  MoveL 2621 to (-2.16, 59.3, -119.45) mm, rotated rx 105.8 ry 33.04 rz -145.95 deg; joints [-4.768, -29.357, 102.728, 146.483, 85.031, 18.435, -295]
  MoveL 2622 to (0.51, 59.77, -119.55) mm, rotated rx 105.8 ry 33.04 rz -145.95 deg; joints [-4.771, -29.24, 102.473, 146.472, 84.917, 18.512, -295]
  MoveL 2623 to (2.52, 60.11, -119.76) mm, rotated rx 105.8 ry 33.04 rz -145.95 deg; joints [-4.779, -29.151, 102.281, 146.459, 84.832, 18.572, -295]
  MoveL 2624 to (4.69, 60.48, -119.96) mm, rotated rx 105.8 ry 33.04 rz -145.95 deg; joints [-4.787, -29.055, 102.073, 146.446, 84.74, 18.636, -295]
  MoveL 2625 to (6.69, 60.8, -120.25) mm, rotated rx 105.8 ry 33.04 rz -145.95 deg; joints [-4.798, -28.966, 101.881, 146.43, 84.657, 18.695, -295]
  MoveL 2626 to (8.64, 61.14, -120.38) mm, rotated rx 105.8 ry 33.04 rz -145.95 deg; joints [-4.803, -28.879, 101.693, 146.42, 84.573, 18.753, -295]
  MoveL 2627 to (10.7, 61.51, -120.39) mm, rotated rx 105.8 ry 33.04 rz -145.95 deg; joints [-4.803, -28.789, 101.495, 146.414, 84.483, 18.813, -295]
  MoveL 2628 to (12.45, 61.78, -120.62) mm, rotated rx 105.8 ry 33.04 rz -145.95 deg; joints [-4.812, -28.709, 101.326, 146.401, 84.41, 18.864, -295]
  Set speed (1000.0 mm/s)
  MoveL 2629 to (33.8, 76.72, -120.62) mm, rotated rx 105.8 ry 33.04 rz -145.95 deg; joints [-4.805, -28.216, 99.114, 146.302, 82.978, 19.821, -295]
  Set speed (1000.0 mm/s)
  MoveL 2630 to (37.55, 71.37, -131.81) mm, rotated rx 105.8 ry 33.04 rz -145.95 deg; joints [-5.233, -27.799, 98.812, 145.891, 83.151, 19.873, -295]
  Set speed (100.0 mm/s)
  MoveL 2631 to (21.02, 59.8, -131.81) mm, rotated rx 105.8 ry 33.04 rz -145.95 deg; joints [-5.244, -28.182, 100.529, 145.963, 84.258, 19.124, -295]
  MoveL 2632 to (18.89, 59.68, -131.81) mm, rotated rx 105.8 ry 33.04 rz -145.95 deg; joints [-5.245, -28.288, 100.733, 145.968, 84.339, 19.069, -295]
  MoveL 2633 to (16.66, 59.58, -131.71) mm, rotated rx 105.8 ry 33.04 rz -145.95 deg; joints [-5.242, -28.4, 100.946, 145.976, 84.423, 19.012, -295]
  MoveL 2634 to (14.32, 59.52, -131.42) mm, rotated rx 105.8 ry 33.04 rz -145.95 deg; joints [-5.231, -28.519, 101.169, 145.992, 84.508, 18.95, -295]
  MoveL 2635 to (12.07, 59.46, -131.07) mm, rotated rx 105.8 ry 33.04 rz -145.95 deg; joints [-5.218, -28.633, 101.383, 146.01, 84.588, 18.891, -295]
  MoveL 2636 to (10, 59.38, -130.88) mm, rotated rx 105.8 ry 33.04 rz -145.95 deg; joints [-5.212, -28.737, 101.579, 146.022, 84.664, 18.837, -295]
  MoveL 2637 to (8.05, 59.28, -130.75) mm, rotated rx 105.8 ry 33.04 rz -145.95 deg; joints [-5.207, -28.833, 101.764, 146.031, 84.736, 18.787, -295]
  MoveL 2638 to (6, 59.18, -130.7) mm, rotated rx 105.8 ry 33.04 rz -145.95 deg; joints [-5.206, -28.935, 101.959, 146.037, 84.813, 18.734, -295]
  MoveL 2639 to (3.87, 59.06, -130.68) mm, rotated rx 105.8 ry 33.04 rz -145.95 deg; joints [-5.205, -29.04, 102.16, 146.042, 84.893, 18.68, -295]
  MoveL 2640 to (1.75, 58.95, -130.56) mm, rotated rx 105.8 ry 33.04 rz -145.95 deg; joints [-5.201, -29.144, 102.361, 146.051, 84.972, 18.625, -295]
  MoveL 2641 to (-0.53, 58.83, -130.3) mm, rotated rx 105.8 ry 33.04 rz -145.95 deg; joints [-5.192, -29.257, 102.576, 146.065, 85.056, 18.565, -295]
  MoveL 2642 to (-2.93, 58.7, -130.11) mm, rotated rx 105.8 ry 33.04 rz -145.95 deg; joints [-5.185, -29.374, 102.802, 146.077, 85.145, 18.503, -295]
  MoveL 2643 to (-5.26, 58.57, -129.91) mm, rotated rx 105.8 ry 33.04 rz -145.95 deg; joints [-5.178, -29.488, 103.021, 146.089, 85.231, 18.442, -295]
  MoveL 2644 to (-7.39, 58.44, -129.8) mm, rotated rx 105.8 ry 33.04 rz -145.95 deg; joints [-5.174, -29.592, 103.221, 146.097, 85.31, 18.388, -295]
  MoveL 2645 to (-11.61, 58.19, -129.52) mm, rotated rx 105.8 ry 33.04 rz -145.95 deg; joints [-5.165, -29.797, 103.616, 146.115, 85.467, 18.279, -295]
  MoveL 2646 to (-13.78, 58.06, -129.46) mm, rotated rx 105.8 ry 33.04 rz -145.95 deg; joints [-5.163, -29.902, 103.819, 146.121, 85.547, 18.224, -295]
  MoveL 2647 to (-15.91, 57.92, -129.24) mm, rotated rx 105.8 ry 33.04 rz -145.95 deg; joints [-5.154, -30.004, 104.017, 146.133, 85.626, 18.168, -295]
  MoveL 2648 to (-18.01, 57.77, -129.08) mm, rotated rx 105.8 ry 33.04 rz -145.95 deg; joints [-5.149, -30.105, 104.214, 146.143, 85.704, 18.114, -295]
  MoveL 2649 to (-20.12, 57.62, -128.89) mm, rotated rx 105.8 ry 33.04 rz -145.95 deg; joints [-5.142, -30.206, 104.41, 146.153, 85.783, 18.059, -295]
  MoveL 2650 to (-22.29, 57.49, -128.8) mm, rotated rx 105.8 ry 33.04 rz -145.95 deg; joints [-5.139, -30.31, 104.611, 146.16, 85.863, 18.004, -295]
  MoveL 2651 to (-24.56, 57.32, -128.67) mm, rotated rx 105.8 ry 33.04 rz -145.95 deg; joints [-5.134, -30.418, 104.822, 146.169, 85.948, 17.945, -295]
  MoveL 2652 to (-26.46, 57.22, -128.61) mm, rotated rx 105.8 ry 33.04 rz -145.95 deg; joints [-5.132, -30.51, 104.998, 146.174, 86.017, 17.898, -295]
  MoveL 2653 to (-26.42, 56.56, -127.73) mm, rotated rx 105.8 ry 33.04 rz -145.95 deg; joints [-5.098, -30.478, 105.002, 146.209, 86.042, 17.87, -295]
  MoveL 2654 to (-26.12, 56.36, -127.32) mm, rotated rx 105.8 ry 33.04 rz -145.95 deg; joints [-5.081, -30.454, 104.977, 146.226, 86.038, 17.867, -295]
  MoveL 2655 to (-26.09, 56.3, -127.04) mm, rotated rx 105.8 ry 33.04 rz -145.95 deg; joints [-5.07, -30.449, 104.975, 146.236, 86.039, 17.863, -295]
  MoveL 2656 to (-26.4, 56.42, -126.92) mm, rotated rx 105.8 ry 33.04 rz -145.95 deg; joints [-5.066, -30.47, 105.002, 146.241, 86.043, 17.859, -295]
  MoveL 2657 to (-26.8, 56.62, -126.86) mm, rotated rx 105.8 ry 33.04 rz -145.95 deg; joints [-5.063, -30.5, 105.037, 146.244, 86.048, 17.855, -295]
  MoveL 2658 to (-27.3, 56.88, -126.83) mm, rotated rx 105.8 ry 33.04 rz -145.95 deg; joints [-5.062, -30.537, 105.08, 146.245, 86.052, 17.852, -295]
  MoveL 2659 to (-27.91, 57.21, -126.79) mm, rotated rx 105.8 ry 33.04 rz -145.95 deg; joints [-5.06, -30.582, 105.132, 146.247, 86.057, 17.848, -295]
  MoveL 2660 to (-28.46, 57.53, -126.76) mm, rotated rx 105.8 ry 33.04 rz -145.95 deg; joints [-5.059, -30.624, 105.179, 146.248, 86.062, 17.845, -295]
  MoveL 2661 to (-28.91, 57.79, -126.76) mm, rotated rx 105.8 ry 33.04 rz -145.95 deg; joints [-5.059, -30.659, 105.218, 146.249, 86.065, 17.843, -295]
  MoveL 2662 to (-29.34, 58.03, -126.75) mm, rotated rx 105.8 ry 33.04 rz -145.95 deg; joints [-5.058, -30.691, 105.254, 146.249, 86.068, 17.84, -295]
  MoveL 2663 to (-30.26, 58.51, -126.67) mm, rotated rx 105.8 ry 33.04 rz -145.95 deg; joints [-5.055, -30.76, 105.333, 146.253, 86.076, 17.833, -295]
  MoveL 2664 to (-30.76, 58.77, -126.62) mm, rotated rx 105.8 ry 33.04 rz -145.95 deg; joints [-5.053, -30.797, 105.376, 146.255, 86.081, 17.83, -295]
  MoveL 2665 to (-31.22, 58.99, -126.55) mm, rotated rx 105.8 ry 33.04 rz -145.95 deg; joints [-5.05, -30.83, 105.416, 146.258, 86.086, 17.825, -295]
  MoveL 2666 to (-31.64, 59.18, -126.48) mm, rotated rx 105.8 ry 33.04 rz -145.95 deg; joints [-5.047, -30.86, 105.452, 146.261, 86.091, 17.821, -295]
  MoveL 2667 to (-32.06, 59.39, -126.42) mm, rotated rx 105.8 ry 33.04 rz -145.95 deg; joints [-5.045, -30.89, 105.488, 146.264, 86.096, 17.817, -295]
  MoveL 2668 to (-32.48, 59.61, -126.39) mm, rotated rx 105.8 ry 33.04 rz -145.95 deg; joints [-5.044, -30.922, 105.525, 146.265, 86.099, 17.814, -295]
  MoveL 2669 to (-32.94, 59.87, -126.37) mm, rotated rx 105.8 ry 33.04 rz -145.95 deg; joints [-5.043, -30.956, 105.564, 146.266, 86.103, 17.812, -295]
  MoveL 2670 to (-36.09, 61.74, -126.37) mm, rotated rx 105.8 ry 33.04 rz -145.95 deg; joints [-5.042, -31.2, 105.831, 146.268, 86.122, 17.799, -295]
  MoveL 2671 to (-37.43, 62.66, -126.39) mm, rotated rx 105.8 ry 33.04 rz -145.95 deg; joints [-5.043, -31.31, 105.942, 146.267, 86.124, 17.798, -295]
  MoveL 2672 to (-37.85, 63.06, -126.42) mm, rotated rx 105.8 ry 33.04 rz -145.95 deg; joints [-5.044, -31.349, 105.976, 146.266, 86.12, 17.801, -295]
  MoveL 2673 to (-38.11, 63.42, -126.45) mm, rotated rx 105.8 ry 33.04 rz -145.95 deg; joints [-5.045, -31.378, 105.995, 146.264, 86.112, 17.807, -295]
  MoveL 2674 to (-38.23, 63.73, -126.49) mm, rotated rx 105.8 ry 33.04 rz -145.95 deg; joints [-5.047, -31.398, 106.003, 146.262, 86.101, 17.814, -295]
  MoveL 2675 to (-38.24, 63.88, -126.52) mm, rotated rx 105.8 ry 33.04 rz -145.95 deg; joints [-5.048, -31.406, 106.002, 146.261, 86.095, 17.819, -295]
  MoveL 2676 to (-38.22, 64.02, -126.54) mm, rotated rx 105.8 ry 33.04 rz -145.95 deg; joints [-5.048, -31.411, 105.999, 146.26, 86.088, 17.824, -295]
  MoveL 2677 to (-38.17, 64.15, -126.57) mm, rotated rx 105.8 ry 33.04 rz -145.95 deg; joints [-5.049, -31.414, 105.993, 146.259, 86.08, 17.829, -295]
  MoveL 2678 to (-38.1, 64.27, -126.6) mm, rotated rx 105.8 ry 33.04 rz -145.95 deg; joints [-5.051, -31.416, 105.985, 146.257, 86.072, 17.835, -295]
  MoveL 2679 to (-37.87, 64.49, -126.66) mm, rotated rx 105.8 ry 33.04 rz -145.95 deg; joints [-5.053, -31.414, 105.962, 146.254, 86.055, 17.847, -295]
  MoveL 2680 to (-37.16, 64.85, -126.79) mm, rotated rx 105.8 ry 33.04 rz -145.95 deg; joints [-5.058, -31.394, 105.893, 146.248, 86.015, 17.876, -295]
  MoveL 2681 to (-36.19, 65.11, -126.93) mm, rotated rx 105.8 ry 33.04 rz -145.95 deg; joints [-5.063, -31.357, 105.801, 146.24, 85.971, 17.907, -295]
  MoveL 2682 to (-33.87, 65.41, -127.2) mm, rotated rx 105.8 ry 33.04 rz -145.95 deg; joints [-5.073, -31.252, 105.586, 146.226, 85.88, 17.971, -295]
  MoveL 2683 to (-31.46, 65.57, -127.44) mm, rotated rx 105.8 ry 33.04 rz -145.95 deg; joints [-5.082, -31.137, 105.364, 146.213, 85.793, 18.032, -295]
  MoveL 2684 to (22.43, 68.71, -132.52) mm, rotated rx 105.8 ry 33.04 rz -145.95 deg; joints [-5.266, -28.487, 100.293, 145.91, 83.814, 19.434, -295]
  MoveL 2685 to (26.26, 68.94, -132.88) mm, rotated rx 105.8 ry 33.04 rz -145.95 deg; joints [-5.279, -28.295, 99.925, 145.887, 83.67, 19.537, -295]
  MoveL 2686 to (30.01, 68.97, -133.3) mm, rotated rx 105.8 ry 33.04 rz -145.95 deg; joints [-5.294, -28.099, 99.565, 145.862, 83.537, 19.633, -295]
  MoveL 2687 to (31.47, 68.71, -133.51) mm, rotated rx 105.8 ry 33.04 rz -145.95 deg; joints [-5.301, -28.01, 99.426, 145.851, 83.497, 19.664, -295]
  MoveL 2688 to (31.97, 68.47, -133.6) mm, rotated rx 105.8 ry 33.04 rz -145.95 deg; joints [-5.305, -27.974, 99.382, 145.847, 83.491, 19.67, -295]
  MoveL 2689 to (32.13, 68.32, -133.65) mm, rotated rx 105.8 ry 33.04 rz -145.95 deg; joints [-5.307, -27.959, 99.368, 145.845, 83.492, 19.67, -295]
  MoveL 2690 to (32.24, 68.14, -133.69) mm, rotated rx 105.8 ry 33.04 rz -145.95 deg; joints [-5.308, -27.946, 99.359, 145.844, 83.496, 19.667, -295]
  MoveL 2691 to (32.29, 67.94, -133.73) mm, rotated rx 105.8 ry 33.04 rz -145.95 deg; joints [-5.31, -27.935, 99.357, 145.843, 83.504, 19.663, -295]
  MoveL 2692 to (32.26, 67.71, -133.76) mm, rotated rx 105.8 ry 33.04 rz -145.95 deg; joints [-5.311, -27.927, 99.362, 145.843, 83.515, 19.655, -295]
  MoveL 2693 to (32.16, 67.45, -133.79) mm, rotated rx 105.8 ry 33.04 rz -145.95 deg; joints [-5.313, -27.921, 99.375, 145.842, 83.53, 19.646, -295]
  MoveL 2694 to (31.99, 67.16, -133.82) mm, rotated rx 105.8 ry 33.04 rz -145.95 deg; joints [-5.314, -27.918, 99.395, 145.843, 83.55, 19.633, -295]
  MoveL 2695 to (30.39, 65.66, -133.87) mm, rotated rx 105.8 ry 33.04 rz -145.95 deg; joints [-5.317, -27.939, 99.566, 145.849, 83.674, 19.549, -295]
  MoveL 2696 to (28.72, 64.39, -133.87) mm, rotated rx 105.8 ry 33.04 rz -145.95 deg; joints [-5.318, -27.974, 99.74, 145.856, 83.79, 19.471, -295]
  MoveL 2697 to (25.42, 62.49, -133.91) mm, rotated rx 105.8 ry 33.04 rz -145.95 deg; joints [-5.322, -28.067, 100.077, 145.867, 83.993, 19.334, -295]
  MoveL 2698 to (22.04, 61.43, -134.02) mm, rotated rx 105.8 ry 33.04 rz -145.95 deg; joints [-5.328, -28.199, 100.412, 145.873, 84.162, 19.221, -295]
  MoveL 2699 to (16, 61.08, -134.32) mm, rotated rx 105.8 ry 33.04 rz -145.95 deg; joints [-5.342, -28.499, 100.99, 145.875, 84.394, 19.068, -295]
  MoveL 2700 to (13.67, 61.43, -134.45) mm, rotated rx 105.8 ry 33.04 rz -145.95 deg; joints [-5.347, -28.636, 101.207, 145.874, 84.462, 19.024, -295]
  MoveL 2701 to (-20.45, 68.13, -136.31) mm, rotated rx 105.8 ry 33.04 rz -145.95 deg; joints [-5.429, -30.689, 104.317, 145.847, 85.349, 18.449, -295]
  MoveL 2702 to (-23.37, 68.69, -136.48) mm, rotated rx 105.8 ry 33.04 rz -145.95 deg; joints [-5.436, -30.864, 104.578, 145.844, 85.422, 18.401, -295]
  MoveL 2703 to (-27.1, 68.94, -136.72) mm, rotated rx 105.8 ry 33.04 rz -145.95 deg; joints [-5.447, -31.066, 104.918, 145.839, 85.537, 18.326, -295]
  MoveL 2704 to (-28.56, 68.71, -136.86) mm, rotated rx 105.8 ry 33.04 rz -145.95 deg; joints [-5.454, -31.131, 105.054, 145.836, 85.598, 18.287, -295]
  MoveL 2705 to (-29.05, 68.47, -136.93) mm, rotated rx 105.8 ry 33.04 rz -145.95 deg; joints [-5.457, -31.145, 105.102, 145.835, 85.626, 18.269, -295]
  MoveL 2706 to (-29.22, 68.32, -136.96) mm, rotated rx 105.8 ry 33.04 rz -145.95 deg; joints [-5.459, -31.147, 105.119, 145.834, 85.639, 18.261, -295]
  MoveL 2707 to (-29.33, 68.14, -137) mm, rotated rx 105.8 ry 33.04 rz -145.95 deg; joints [-5.46, -31.144, 105.131, 145.833, 85.651, 18.253, -295]
  MoveL 2708 to (-29.37, 67.93, -137.03) mm, rotated rx 105.8 ry 33.04 rz -145.95 deg; joints [-5.462, -31.137, 105.137, 145.832, 85.662, 18.246, -295]
  MoveL 2709 to (-29.34, 67.7, -137.07) mm, rotated rx 105.8 ry 33.04 rz -145.95 deg; joints [-5.463, -31.126, 105.137, 145.831, 85.672, 18.24, -295]
  MoveL 2710 to (-29.24, 67.44, -137.1) mm, rotated rx 105.8 ry 33.04 rz -145.95 deg; joints [-5.465, -31.109, 105.131, 145.83, 85.681, 18.234, -295]
  MoveL 2711 to (-29.06, 67.14, -137.14) mm, rotated rx 105.8 ry 33.04 rz -145.95 deg; joints [-5.466, -31.087, 105.118, 145.829, 85.689, 18.23, -295]
  MoveL 2712 to (-27.45, 65.66, -137.26) mm, rotated rx 105.8 ry 33.04 rz -145.95 deg; joints [-5.471, -30.939, 104.987, 145.825, 85.704, 18.221, -295]
  MoveL 2713 to (-27.03, 65.35, -137.28) mm, rotated rx 105.8 ry 33.04 rz -145.95 deg; joints [-5.472, -30.904, 104.952, 145.824, 85.704, 18.221, -295]
  MoveL 2714 to (-26.65, 65.1, -137.33) mm, rotated rx 105.8 ry 33.04 rz -145.95 deg; joints [-5.474, -30.873, 104.92, 145.822, 85.703, 18.222, -295]
  MoveL 2715 to (-26.27, 64.88, -137.4) mm, rotated rx 105.8 ry 33.04 rz -145.95 deg; joints [-5.477, -30.843, 104.888, 145.819, 85.701, 18.225, -295]
  MoveL 2716 to (-25.9, 64.64, -137.46) mm, rotated rx 105.8 ry 33.04 rz -145.95 deg; joints [-5.479, -30.814, 104.856, 145.817, 85.7, 18.226, -295]
  MoveL 2717 to (-25.51, 64.37, -137.49) mm, rotated rx 105.8 ry 33.04 rz -145.95 deg; joints [-5.48, -30.783, 104.824, 145.815, 85.699, 18.227, -295]
  MoveL 2718 to (-21.81, 61.5, -137.5) mm, rotated rx 105.8 ry 33.04 rz -145.95 deg; joints [-5.481, -30.466, 104.516, 145.815, 85.706, 18.223, -295]
  MoveL 2719 to (-21.46, 61.24, -137.52) mm, rotated rx 105.8 ry 33.04 rz -145.95 deg; joints [-5.482, -30.437, 104.486, 145.814, 85.706, 18.223, -295]
  MoveL 2720 to (-21.08, 60.95, -137.53) mm, rotated rx 105.8 ry 33.04 rz -145.95 deg; joints [-5.482, -30.404, 104.454, 145.814, 85.707, 18.223, -295]
  MoveL 2721 to (-20.26, 60.32, -137.53) mm, rotated rx 105.8 ry 33.04 rz -145.95 deg; joints [-5.482, -30.335, 104.386, 145.814, 85.708, 18.222, -295]
  MoveL 2722 to (-19.8, 59.97, -137.54) mm, rotated rx 105.8 ry 33.04 rz -145.95 deg; joints [-5.483, -30.296, 104.347, 145.814, 85.708, 18.222, -295]
  MoveL 2723 to (-19.31, 59.63, -137.56) mm, rotated rx 105.8 ry 33.04 rz -145.95 deg; joints [-5.483, -30.255, 104.305, 145.813, 85.707, 18.223, -295]
  MoveL 2724 to (-18.74, 59.28, -137.59) mm, rotated rx 105.8 ry 33.04 rz -145.95 deg; joints [-5.484, -30.211, 104.257, 145.812, 85.704, 18.226, -295]
  MoveL 2725 to (-18.14, 59, -137.61) mm, rotated rx 105.8 ry 33.04 rz -145.95 deg; joints [-5.485, -30.168, 104.204, 145.81, 85.696, 18.231, -295]
  MoveL 2726 to (-17.53, 58.78, -137.63) mm, rotated rx 105.8 ry 33.04 rz -145.95 deg; joints [-5.486, -30.127, 104.15, 145.809, 85.685, 18.238, -295]
  MoveL 2727 to (-18.63, 59.49, -138.61) mm, rotated rx 105.8 ry 33.04 rz -145.95 deg; joints [-5.524, -30.215, 104.243, 145.772, 85.695, 18.245, -295]
  MoveL 2728 to (-17.31, 59.72, -139.03) mm, rotated rx 105.8 ry 33.04 rz -145.95 deg; joints [-5.541, -30.158, 104.118, 145.753, 85.642, 18.287, -295]
  MoveL 2729 to (-15.82, 59.83, -139.35) mm, rotated rx 105.8 ry 33.04 rz -145.95 deg; joints [-5.552, -30.087, 103.979, 145.738, 85.587, 18.328, -295]
  MoveL 2730 to (-14.12, 59.85, -139.59) mm, rotated rx 105.8 ry 33.04 rz -145.95 deg; joints [-5.561, -30.001, 103.821, 145.727, 85.529, 18.37, -295]
  MoveL 2731 to (-11.99, 59.75, -139.81) mm, rotated rx 105.8 ry 33.04 rz -145.95 deg; joints [-5.568, -29.887, 103.624, 145.716, 85.462, 18.419, -295]
  MoveL 2732 to (-9.86, 59.62, -139.92) mm, rotated rx 105.8 ry 33.04 rz -145.95 deg; joints [-5.572, -29.772, 103.428, 145.709, 85.395, 18.466, -295]
  MoveL 2733 to (-7.73, 59.49, -140.03) mm, rotated rx 105.8 ry 33.04 rz -145.95 deg; joints [-5.575, -29.657, 103.231, 145.702, 85.328, 18.513, -295]
  MoveL 2734 to (-5.6, 59.37, -140.26) mm, rotated rx 105.8 ry 33.04 rz -145.95 deg; joints [-5.583, -29.543, 103.033, 145.69, 85.261, 18.562, -295]
  MoveL 2735 to (-3.47, 59.23, -140.38) mm, rotated rx 105.8 ry 33.04 rz -145.95 deg; joints [-5.587, -29.427, 102.836, 145.683, 85.193, 18.609, -295]
  MoveL 2736 to (-1.34, 59.1, -140.61) mm, rotated rx 105.8 ry 33.04 rz -145.95 deg; joints [-5.595, -29.312, 102.638, 145.671, 85.126, 18.658, -295]
  MoveL 2737 to (0.79, 58.95, -140.73) mm, rotated rx 105.8 ry 33.04 rz -145.95 deg; joints [-5.599, -29.196, 102.44, 145.663, 85.059, 18.705, -295]
  MoveL 2738 to (2.92, 58.81, -140.84) mm, rotated rx 105.8 ry 33.04 rz -145.95 deg; joints [-5.602, -29.08, 102.242, 145.656, 84.992, 18.752, -295]
  MoveL 2739 to (5.05, 58.66, -141.08) mm, rotated rx 105.8 ry 33.04 rz -145.95 deg; joints [-5.61, -28.964, 102.043, 145.644, 84.925, 18.801, -295]
  MoveL 2740 to (7.08, 58.5, -141.18) mm, rotated rx 105.8 ry 33.04 rz -145.95 deg; joints [-5.614, -28.852, 101.853, 145.637, 84.861, 18.846, -295]
  MoveL 2741 to (9.06, 58.35, -141.39) mm, rotated rx 105.8 ry 33.04 rz -145.95 deg; joints [-5.621, -28.743, 101.668, 145.626, 84.8, 18.891, -295]
  MoveL 2742 to (11.43, 58.19, -141.55) mm, rotated rx 105.8 ry 33.04 rz -145.95 deg; joints [-5.626, -28.613, 101.446, 145.616, 84.724, 18.945, -295]
  MoveL 2743 to (14.14, 57.96, -141.64) mm, rotated rx 105.8 ry 33.04 rz -145.95 deg; joints [-5.628, -28.463, 101.191, 145.609, 84.639, 19.004, -295]
  MoveL 2744 to (16.21, 57.81, -141.71) mm, rotated rx 105.8 ry 33.04 rz -145.95 deg; joints [-5.629, -28.349, 100.997, 145.603, 84.572, 19.05, -295]
  MoveL 2745 to (18.13, 57.67, -141.83) mm, rotated rx 105.8 ry 33.04 rz -145.95 deg; joints [-5.634, -28.243, 100.816, 145.595, 84.511, 19.094, -295]
  MoveL 2746 to (20.11, 57.52, -141.94) mm, rotated rx 105.8 ry 33.04 rz -145.95 deg; joints [-5.637, -28.134, 100.629, 145.587, 84.448, 19.139, -295]
  MoveL 2747 to (22.05, 57.37, -142.05) mm, rotated rx 105.8 ry 33.04 rz -145.95 deg; joints [-5.64, -28.026, 100.445, 145.58, 84.386, 19.183, -295]
  MoveL 2748 to (24.11, 57.21, -142.12) mm, rotated rx 105.8 ry 33.04 rz -145.95 deg; joints [-5.642, -27.912, 100.25, 145.574, 84.319, 19.229, -295]
  MoveL 2749 to (26.32, 57.03, -142.22) mm, rotated rx 105.8 ry 33.04 rz -145.95 deg; joints [-5.644, -27.789, 100.04, 145.566, 84.248, 19.279, -295]
  MoveL 2750 to (28.72, 56.81, -142.48) mm, rotated rx 105.8 ry 33.04 rz -145.95 deg; joints [-5.653, -27.654, 99.813, 145.552, 84.173, 19.334, -295]
  MoveL 2751 to (30.94, 57.13, -143.46) mm, rotated rx 105.8 ry 33.04 rz -145.95 deg; joints [-5.69, -27.551, 99.595, 145.51, 84.084, 19.409, -295]
  MoveL 2752 to (29.94, 56.57, -143.95) mm, rotated rx 105.8 ry 33.04 rz -145.95 deg; joints [-5.709, -27.58, 99.696, 145.495, 84.147, 19.373, -295]
  MoveL 2753 to (29.42, 56.28, -144.26) mm, rotated rx 105.8 ry 33.04 rz -145.95 deg; joints [-5.722, -27.595, 99.749, 145.485, 84.181, 19.354, -295]
  MoveL 2754 to (29.34, 56.23, -144.41) mm, rotated rx 105.8 ry 33.04 rz -145.95 deg; joints [-5.728, -27.597, 99.757, 145.48, 84.187, 19.352, -295]
  MoveL 2755 to (29.64, 56.39, -144.45) mm, rotated rx 105.8 ry 33.04 rz -145.95 deg; joints [-5.729, -27.588, 99.726, 145.477, 84.169, 19.365, -295]
  MoveL 2756 to (30.05, 56.62, -144.46) mm, rotated rx 105.8 ry 33.04 rz -145.95 deg; joints [-5.729, -27.576, 99.684, 145.475, 84.144, 19.382, -295]
  MoveL 2757 to (30.47, 56.84, -144.5) mm, rotated rx 105.8 ry 33.04 rz -145.95 deg; joints [-5.73, -27.563, 99.641, 145.473, 84.12, 19.4, -295]
  MoveL 2758 to (30.88, 57.03, -144.56) mm, rotated rx 105.8 ry 33.04 rz -145.95 deg; joints [-5.732, -27.55, 99.6, 145.469, 84.097, 19.416, -295]
  MoveL 2759 to (31.29, 57.23, -144.6) mm, rotated rx 105.8 ry 33.04 rz -145.95 deg; joints [-5.733, -27.537, 99.558, 145.466, 84.073, 19.433, -295]
  MoveL 2760 to (31.73, 57.47, -144.62) mm, rotated rx 105.8 ry 33.04 rz -145.95 deg; joints [-5.733, -27.524, 99.514, 145.464, 84.047, 19.451, -295]
  MoveL 2761 to (34, 58.77, -144.62) mm, rotated rx 105.8 ry 33.04 rz -145.95 deg; joints [-5.731, -27.46, 99.281, 145.456, 83.908, 19.547, -295]
  MoveL 2762 to (34.4, 58.98, -144.64) mm, rotated rx 105.8 ry 33.04 rz -145.95 deg; joints [-5.731, -27.448, 99.239, 145.454, 83.884, 19.563, -295]
  MoveL 2763 to (34.75, 59.15, -144.67) mm, rotated rx 105.8 ry 33.04 rz -145.95 deg; joints [-5.732, -27.437, 99.204, 145.452, 83.864, 19.577, -295]
  MoveL 2764 to (35.16, 59.37, -144.69) mm, rotated rx 105.8 ry 33.04 rz -145.95 deg; joints [-5.733, -27.424, 99.162, 145.449, 83.84, 19.594, -295]
  MoveL 2765 to (35.68, 59.65, -144.71) mm, rotated rx 105.8 ry 33.04 rz -145.95 deg; joints [-5.733, -27.409, 99.109, 145.447, 83.809, 19.616, -295]
  MoveL 2766 to (36.33, 59.98, -144.77) mm, rotated rx 105.8 ry 33.04 rz -145.95 deg; joints [-5.735, -27.388, 99.043, 145.442, 83.772, 19.642, -295]
  MoveL 2767 to (36.88, 60.27, -144.8) mm, rotated rx 105.8 ry 33.04 rz -145.95 deg; joints [-5.735, -27.372, 98.987, 145.439, 83.739, 19.665, -295]
  MoveL 2768 to (37.34, 60.53, -144.8) mm, rotated rx 105.8 ry 33.04 rz -145.95 deg; joints [-5.735, -27.358, 98.939, 145.438, 83.711, 19.685, -295]
  MoveL 2769 to (38.71, 61.31, -144.8) mm, rotated rx 105.8 ry 33.04 rz -145.95 deg; joints [-5.734, -27.319, 98.798, 145.433, 83.627, 19.742, -295]
  MoveL 2770 to (41.37, 62.49, -145.14) mm, rotated rx 105.8 ry 33.04 rz -145.95 deg; joints [-5.744, -27.228, 98.527, 145.411, 83.481, 19.848, -295]
  MoveL 2771 to (42.63, 62.79, -145.57) mm, rotated rx 105.8 ry 33.04 rz -145.95 deg; joints [-5.76, -27.173, 98.4, 145.391, 83.425, 19.893, -295]
  MoveL 2772 to (43.84, 62.89, -146.17) mm, rotated rx 105.8 ry 33.04 rz -145.95 deg; joints [-5.782, -27.113, 98.28, 145.365, 83.379, 19.933, -295]
  MoveL 2773 to (46.13, 62.5, -147.88) mm, rotated rx 105.8 ry 33.04 rz -145.95 deg; joints [-5.845, -26.975, 98.059, 145.298, 83.322, 19.998, -295]
  MoveL 2774 to (48.23, 61.33, -150.28) mm, rotated rx 105.8 ry 33.04 rz -145.95 deg; joints [-5.936, -26.814, 97.863, 145.207, 83.31, 20.043, -295]
  MoveL 2775 to (49.62, 59.81, -152.67) mm, rotated rx 105.8 ry 33.04 rz -145.95 deg; joints [-6.026, -26.677, 97.739, 145.119, 83.338, 20.059, -295]
  MoveL 2776 to (49.86, 59.08, -153.61) mm, rotated rx 105.8 ry 33.04 rz -145.95 deg; joints [-6.062, -26.634, 97.722, 145.086, 83.366, 20.054, -295]
  MoveL 2777 to (49.78, 58.38, -154.38) mm, rotated rx 105.8 ry 33.04 rz -145.95 deg; joints [-6.092, -26.609, 97.735, 145.059, 83.403, 20.039, -295]
  MoveL 2778 to (49.62, 58.03, -154.7) mm, rotated rx 105.8 ry 33.04 rz -145.95 deg; joints [-6.105, -26.602, 97.754, 145.049, 83.425, 20.029, -295]
  MoveL 2779 to (49.39, 57.69, -154.98) mm, rotated rx 105.8 ry 33.04 rz -145.95 deg; joints [-6.116, -26.601, 97.779, 145.04, 83.45, 20.016, -295]
  MoveL 2780 to (48.7, 57.03, -155.41) mm, rotated rx 105.8 ry 33.04 rz -145.95 deg; joints [-6.133, -26.61, 97.853, 145.027, 83.506, 19.983, -295]
  MoveL 2781 to (47.69, 56.39, -155.67) mm, rotated rx 105.8 ry 33.04 rz -145.95 deg; joints [-6.144, -26.636, 97.957, 145.021, 83.572, 19.941, -295]
  MoveL 2782 to (46.38, 55.78, -155.75) mm, rotated rx 105.8 ry 33.04 rz -145.95 deg; joints [-6.149, -26.68, 98.092, 145.022, 83.647, 19.89, -295]
  MoveL 2783 to (45.89, 55.58, -155.75) mm, rotated rx 105.8 ry 33.04 rz -145.95 deg; joints [-6.149, -26.697, 98.141, 145.024, 83.673, 19.872, -295]
  MoveL 2784 to (45.48, 55.45, -155.7) mm, rotated rx 105.8 ry 33.04 rz -145.95 deg; joints [-6.148, -26.714, 98.183, 145.027, 83.694, 19.856, -295]
  MoveL 2785 to (45.06, 55.32, -155.64) mm, rotated rx 105.8 ry 33.04 rz -145.95 deg; joints [-6.146, -26.73, 98.225, 145.031, 83.715, 19.841, -295]
  MoveL 2786 to (44.61, 55.16, -155.6) mm, rotated rx 105.8 ry 33.04 rz -145.95 deg; joints [-6.145, -26.747, 98.27, 145.033, 83.738, 19.825, -295]
  MoveL 2787 to (44.15, 54.99, -155.58) mm, rotated rx 105.8 ry 33.04 rz -145.95 deg; joints [-6.145, -26.764, 98.317, 145.035, 83.762, 19.808, -295]
  MoveL 2788 to (43.65, 54.79, -155.58) mm, rotated rx 105.8 ry 33.04 rz -145.95 deg; joints [-6.145, -26.782, 98.368, 145.037, 83.789, 19.789, -295]
  MoveL 2789 to (43.17, 54.59, -155.58) mm, rotated rx 105.8 ry 33.04 rz -145.95 deg; joints [-6.146, -26.799, 98.417, 145.038, 83.815, 19.771, -295]
  MoveL 2790 to (42.71, 54.38, -155.59) mm, rotated rx 105.8 ry 33.04 rz -145.95 deg; joints [-6.147, -26.815, 98.464, 145.039, 83.841, 19.753, -295]
  MoveL 2791 to (42.25, 54.18, -155.6) mm, rotated rx 105.8 ry 33.04 rz -145.95 deg; joints [-6.148, -26.831, 98.51, 145.04, 83.866, 19.736, -295]
  MoveL 2792 to (41.82, 54.02, -155.58) mm, rotated rx 105.8 ry 33.04 rz -145.95 deg; joints [-6.148, -26.847, 98.554, 145.042, 83.889, 19.719, -295]
  MoveL 2793 to (41.38, 53.86, -155.54) mm, rotated rx 105.8 ry 33.04 rz -145.95 deg; joints [-6.146, -26.863, 98.598, 145.045, 83.911, 19.703, -295]
  MoveL 2794 to (40.87, 53.69, -155.49) mm, rotated rx 105.8 ry 33.04 rz -145.95 deg; joints [-6.145, -26.883, 98.65, 145.048, 83.938, 19.684, -295]
  MoveL 2795 to (40.2, 53.46, -155.44) mm, rotated rx 105.8 ry 33.04 rz -145.95 deg; joints [-6.144, -26.908, 98.717, 145.052, 83.971, 19.66, -295]
  MoveL 2796 to (39.6, 53.23, -155.42) mm, rotated rx 105.8 ry 33.04 rz -145.95 deg; joints [-6.144, -26.93, 98.778, 145.055, 84.003, 19.638, -295]
  MoveL 2797 to (37.18, 52.23, -155.42) mm, rotated rx 105.8 ry 33.04 rz -145.95 deg; joints [-6.146, -27.015, 99.022, 145.061, 84.135, 19.546, -295]
  MoveL 2798 to (36.59, 52.01, -155.38) mm, rotated rx 105.8 ry 33.04 rz -145.95 deg; joints [-6.146, -27.036, 99.081, 145.064, 84.165, 19.525, -295]
  MoveL 2799 to (36.07, 51.82, -155.32) mm, rotated rx 105.8 ry 33.04 rz -145.95 deg; joints [-6.144, -27.056, 99.134, 145.068, 84.192, 19.505, -295]
  MoveL 2800 to (35.87, 51.76, -155.17) mm, rotated rx 105.8 ry 33.04 rz -145.95 deg; joints [-6.139, -27.064, 99.154, 145.074, 84.201, 19.497, -295]
  MoveL 2801 to (35.98, 51.8, -154.91) mm, rotated rx 105.8 ry 33.04 rz -145.95 deg; joints [-6.128, -27.059, 99.143, 145.083, 84.194, 19.498, -295]
  MoveL 2802 to (36.42, 51.94, -154.5) mm, rotated rx 105.8 ry 33.04 rz -145.95 deg; joints [-6.112, -27.043, 99.101, 145.098, 84.17, 19.509, -295]
  MoveL 2803 to (35.75, 52.72, -153.7) mm, rotated rx 105.8 ry 33.04 rz -145.95 deg; joints [-6.082, -27.111, 99.159, 145.127, 84.156, 19.507, -295]
  MoveL 2804 to (33.82, 53.17, -153.48) mm, rotated rx 105.8 ry 33.04 rz -145.95 deg; joints [-6.074, -27.231, 99.341, 145.138, 84.206, 19.469, -295]
  MoveL 2805 to (31.86, 53.6, -153.32) mm, rotated rx 105.8 ry 33.04 rz -145.95 deg; joints [-6.07, -27.352, 99.525, 145.146, 84.257, 19.431, -295]
  MoveL 2806 to (29.85, 54.03, -153.17) mm, rotated rx 105.8 ry 33.04 rz -145.95 deg; joints [-6.065, -27.476, 99.714, 145.154, 84.31, 19.393, -295]
  MoveL 2807 to (28.02, 54.44, -152.88) mm, rotated rx 105.8 ry 33.04 rz -145.95 deg; joints [-6.055, -27.589, 99.886, 145.167, 84.357, 19.356, -295]
  MoveL 2808 to (25.95, 54.89, -152.69) mm, rotated rx 105.8 ry 33.04 rz -145.95 deg; joints [-6.049, -27.715, 100.08, 145.177, 84.411, 19.316, -295]
  MoveL 2809 to (23.79, 55.35, -152.51) mm, rotated rx 105.8 ry 33.04 rz -145.95 deg; joints [-6.043, -27.848, 100.282, 145.187, 84.467, 19.275, -295]
  MoveL 2810 to (21.59, 55.81, -152.42) mm, rotated rx 105.8 ry 33.04 rz -145.95 deg; joints [-6.041, -27.982, 100.487, 145.192, 84.525, 19.234, -295]
  MoveL 2811 to (18.92, 56.36, -152.33) mm, rotated rx 105.8 ry 33.04 rz -145.95 deg; joints [-6.039, -28.145, 100.736, 145.199, 84.595, 19.184, -295]
  MoveL 2812 to (17, 56.75, -152.22) mm, rotated rx 105.8 ry 33.04 rz -145.95 deg; joints [-6.036, -28.261, 100.914, 145.205, 84.645, 19.148, -295]
  MoveL 2813 to (15.21, 57.11, -152.01) mm, rotated rx 105.8 ry 33.04 rz -145.95 deg; joints [-6.029, -28.37, 101.081, 145.215, 84.692, 19.113, -295]
  MoveL 2814 to (13.23, 57.51, -151.82) mm, rotated rx 105.8 ry 33.04 rz -145.95 deg; joints [-6.023, -28.49, 101.264, 145.225, 84.743, 19.075, -295]
  MoveL 2815 to (11.14, 57.93, -151.7) mm, rotated rx 105.8 ry 33.04 rz -145.95 deg; joints [-6.02, -28.616, 101.458, 145.231, 84.797, 19.036, -295]
  MoveL 2816 to (9.06, 58.34, -151.52) mm, rotated rx 105.8 ry 33.04 rz -145.95 deg; joints [-6.014, -28.741, 101.65, 145.24, 84.851, 18.996, -295]
  MoveL 2817 to (6.99, 58.75, -151.4) mm, rotated rx 105.8 ry 33.04 rz -145.95 deg; joints [-6.011, -28.866, 101.841, 145.247, 84.905, 18.957, -295]
  MoveL 2818 to (4.85, 59.17, -151.22) mm, rotated rx 105.8 ry 33.04 rz -145.95 deg; joints [-6.005, -28.995, 102.038, 145.256, 84.961, 18.917, -295]
  MoveL 2819 to (2.76, 59.57, -151.1) mm, rotated rx 105.8 ry 33.04 rz -145.95 deg; joints [-6.002, -29.121, 102.231, 145.263, 85.015, 18.878, -295]
  MoveL 2820 to (0.66, 59.96, -150.87) mm, rotated rx 105.8 ry 33.04 rz -145.95 deg; joints [-5.994, -29.246, 102.424, 145.274, 85.069, 18.837, -295]
  MoveL 2821 to (-1.44, 60.37, -150.76) mm, rotated rx 105.8 ry 33.04 rz -145.95 deg; joints [-5.991, -29.372, 102.616, 145.28, 85.124, 18.798, -295]
  MoveL 2822 to (-3.54, 60.76, -150.64) mm, rotated rx 105.8 ry 33.04 rz -145.95 deg; joints [-5.987, -29.497, 102.808, 145.286, 85.178, 18.76, -295]
  MoveL 2823 to (-5.64, 61.14, -150.42) mm, rotated rx 105.8 ry 33.04 rz -145.95 deg; joints [-5.98, -29.622, 103.001, 145.297, 85.232, 18.719, -295]
  MoveL 2824 to (-7.56, 61.43, -150.21) mm, rotated rx 105.8 ry 33.04 rz -145.95 deg; joints [-5.973, -29.733, 103.176, 145.306, 85.284, 18.681, -295]
  MoveL 2825 to (-9.31, 61.63, -149.92) mm, rotated rx 105.8 ry 33.04 rz -145.95 deg; joints [-5.963, -29.832, 103.337, 145.319, 85.334, 18.643, -295]
  MoveL 2826 to (-10.93, 61.74, -149.52) mm, rotated rx 105.8 ry 33.04 rz -145.95 deg; joints [-5.948, -29.92, 103.488, 145.337, 85.383, 18.604, -295]
  MoveL 2827 to (-9.67, 60.96, -148.59) mm, rotated rx 105.8 ry 33.04 rz -145.95 deg; joints [-5.911, -29.821, 103.381, 145.372, 85.37, 18.599, -295]
  MoveL 2828 to (-10.2, 61.18, -148.58) mm, rotated rx 105.8 ry 33.04 rz -145.95 deg; joints [-5.911, -29.858, 103.428, 145.373, 85.378, 18.594, -295]
  MoveL 2829 to (-10.68, 61.42, -148.56) mm, rotated rx 105.8 ry 33.04 rz -145.95 deg; joints [-5.91, -29.893, 103.469, 145.374, 85.384, 18.59, -295]
  MoveL 2830 to (-11.07, 61.68, -148.5) mm, rotated rx 105.8 ry 33.04 rz -145.95 deg; joints [-5.908, -29.925, 103.504, 145.376, 85.386, 18.588, -295]
  MoveL 2831 to (-11.44, 61.93, -148.43) mm, rotated rx 105.8 ry 33.04 rz -145.95 deg; joints [-5.906, -29.955, 103.535, 145.379, 85.386, 18.587, -295]
  MoveL 2832 to (-11.8, 62.23, -148.38) mm, rotated rx 105.8 ry 33.04 rz -145.95 deg; joints [-5.904, -29.986, 103.565, 145.381, 85.385, 18.587, -295]
  MoveL 2833 to (-12.16, 62.56, -148.35) mm, rotated rx 105.8 ry 33.04 rz -145.95 deg; joints [-5.903, -30.019, 103.595, 145.382, 85.382, 18.588, -295]
  MoveL 2834 to (-12.54, 62.92, -148.33) mm, rotated rx 105.8 ry 33.04 rz -145.95 deg; joints [-5.902, -30.055, 103.626, 145.382, 85.378, 18.591, -295]
  MoveL 2835 to (-12.91, 63.29, -148.33) mm, rotated rx 105.8 ry 33.04 rz -145.95 deg; joints [-5.902, -30.09, 103.656, 145.382, 85.374, 18.594, -295]
  MoveL 2836 to (-13.24, 63.62, -148.32) mm, rotated rx 105.8 ry 33.04 rz -145.95 deg; joints [-5.901, -30.121, 103.684, 145.382, 85.371, 18.596, -295]
  MoveL 2837 to (-13.56, 63.9, -148.3) mm, rotated rx 105.8 ry 33.04 rz -145.95 deg; joints [-5.9, -30.15, 103.71, 145.383, 85.368, 18.597, -295]
  MoveL 2838 to (-13.91, 64.24, -148.28) mm, rotated rx 105.8 ry 33.04 rz -145.95 deg; joints [-5.9, -30.183, 103.738, 145.383, 85.365, 18.599, -295]
  MoveL 2839 to (-14.27, 64.61, -148.28) mm, rotated rx 105.8 ry 33.04 rz -145.95 deg; joints [-5.9, -30.218, 103.768, 145.383, 85.36, 18.602, -295]
  MoveL 2840 to (-14.71, 65.04, -148.26) mm, rotated rx 105.8 ry 33.04 rz -145.95 deg; joints [-5.899, -30.259, 103.804, 145.384, 85.356, 18.605, -295]
  MoveL 2841 to (-15.22, 65.51, -148.22) mm, rotated rx 105.8 ry 33.04 rz -145.95 deg; joints [-5.897, -30.306, 103.845, 145.385, 85.351, 18.608, -295]
  MoveL 2842 to (-15.65, 65.94, -148.2) mm, rotated rx 105.8 ry 33.04 rz -145.95 deg; joints [-5.897, -30.347, 103.881, 145.386, 85.346, 18.611, -295]
  MoveL 2843 to (-16.12, 66.38, -148.17) mm, rotated rx 105.8 ry 33.04 rz -145.95 deg; joints [-5.896, -30.39, 103.919, 145.386, 85.342, 18.614, -295]
  MoveL 2844 to (-16.64, 66.86, -148.13) mm, rotated rx 105.8 ry 33.04 rz -145.95 deg; joints [-5.894, -30.438, 103.962, 145.388, 85.338, 18.616, -295]
  MoveL 2845 to (-17.07, 67.27, -148.12) mm, rotated rx 105.8 ry 33.04 rz -145.95 deg; joints [-5.894, -30.478, 103.996, 145.388, 85.333, 18.619, -295]
  MoveL 2846 to (-17.45, 67.66, -148.12) mm, rotated rx 105.8 ry 33.04 rz -145.95 deg; joints [-5.893, -30.515, 104.027, 145.388, 85.328, 18.622, -295]
  MoveL 2847 to (-18.56, 68.77, -148.12) mm, rotated rx 105.8 ry 33.04 rz -145.95 deg; joints [-5.893, -30.621, 104.117, 145.387, 85.315, 18.632, -295]
  MoveL 2848 to (-19.53, 69.85, -148.2) mm, rotated rx 105.8 ry 33.04 rz -145.95 deg; joints [-5.897, -30.718, 104.193, 145.383, 85.298, 18.644, -295]
  MoveL 2849 to (-20.21, 70.83, -148.46) mm, rotated rx 105.8 ry 33.04 rz -145.95 deg; joints [-5.906, -30.795, 104.244, 145.372, 85.278, 18.662, -295]
  MoveL 2850 to (-20.59, 71.7, -148.88) mm, rotated rx 105.8 ry 33.04 rz -145.95 deg; joints [-5.923, -30.854, 104.268, 145.355, 85.252, 18.685, -295]
  MoveL 2851 to (-20.67, 72.11, -149.15) mm, rotated rx 105.8 ry 33.04 rz -145.95 deg; joints [-5.933, -30.875, 104.27, 145.344, 85.238, 18.699, -295]
  MoveL 2852 to (-20.68, 72.48, -149.47) mm, rotated rx 105.8 ry 33.04 rz -145.95 deg; joints [-5.945, -30.892, 104.266, 145.331, 85.223, 18.714, -295]
  MoveL 2853 to (-20.48, 73.16, -150.23) mm, rotated rx 105.8 ry 33.04 rz -145.95 deg; joints [-5.975, -30.911, 104.238, 145.3, 85.188, 18.748, -295]
  MoveL 2854 to (-19.98, 73.73, -151.16) mm, rotated rx 105.8 ry 33.04 rz -145.95 deg; joints [-6.01, -30.911, 104.183, 145.262, 85.15, 18.787, -295]
  MoveL 2855 to (-18.11, 74.59, -153.52) mm, rotated rx 105.8 ry 33.04 rz -145.95 deg; joints [-6.101, -30.851, 103.995, 145.167, 85.06, 18.882, -295]
  MoveL 2856 to (-15.72, 74.84, -155.88) mm, rotated rx 105.8 ry 33.04 rz -145.95 deg; joints [-6.192, -30.738, 103.766, 145.073, 84.979, 18.97, -295]
  MoveL 2857 to (-13.46, 74.3, -157.57) mm, rotated rx 105.8 ry 33.04 rz -145.95 deg; joints [-6.256, -30.597, 103.559, 145.006, 84.936, 19.024, -295]
  MoveL 2858 to (-12.38, 73.73, -158.16) mm, rotated rx 105.8 ry 33.04 rz -145.95 deg; joints [-6.279, -30.516, 103.464, 144.984, 84.929, 19.037, -295]
  MoveL 2859 to (-11.34, 72.97, -158.58) mm, rotated rx 105.8 ry 33.04 rz -145.95 deg; joints [-6.295, -30.429, 103.375, 144.968, 84.93, 19.042, -295]
  MoveL 2860 to (-9.34, 70.84, -158.92) mm, rotated rx 105.8 ry 33.04 rz -145.95 deg; joints [-6.308, -30.233, 103.215, 144.957, 84.961, 19.025, -295]
  MoveL 2861 to (-6.8, 67.51, -158.92) mm, rotated rx 105.8 ry 33.04 rz -145.95 deg; joints [-6.309, -29.957, 103.017, 144.96, 85.025, 18.98, -295]
  MoveL 2862 to (-6.45, 67.09, -158.94) mm, rotated rx 105.8 ry 33.04 rz -145.95 deg; joints [-6.309, -29.921, 102.99, 144.96, 85.033, 18.975, -295]
  MoveL 2863 to (-6.11, 66.68, -158.98) mm, rotated rx 105.8 ry 33.04 rz -145.95 deg; joints [-6.311, -29.886, 102.962, 144.959, 85.039, 18.971, -295]
  MoveL 2864 to (-5.76, 66.29, -159.04) mm, rotated rx 105.8 ry 33.04 rz -145.95 deg; joints [-6.313, -29.85, 102.934, 144.957, 85.045, 18.968, -295]
  MoveL 2865 to (-5.4, 65.92, -159.12) mm, rotated rx 105.8 ry 33.04 rz -145.95 deg; joints [-6.317, -29.815, 102.904, 144.954, 85.05, 18.965, -295]
  MoveL 2866 to (-5.05, 65.55, -159.2) mm, rotated rx 105.8 ry 33.04 rz -145.95 deg; joints [-6.32, -29.781, 102.876, 144.951, 85.055, 18.963, -295]
  MoveL 2867 to (-4.73, 65.18, -159.24) mm, rotated rx 105.8 ry 33.04 rz -145.95 deg; joints [-6.321, -29.749, 102.85, 144.95, 85.061, 18.959, -295]
  MoveL 2868 to (-4.43, 64.8, -159.25) mm, rotated rx 105.8 ry 33.04 rz -145.95 deg; joints [-6.322, -29.717, 102.826, 144.95, 85.068, 18.955, -295]
  MoveL 2869 to (-4.11, 64.39, -159.25) mm, rotated rx 105.8 ry 33.04 rz -145.95 deg; joints [-6.322, -29.683, 102.801, 144.95, 85.076, 18.949, -295]
  MoveL 2870 to (-3.72, 63.9, -159.29) mm, rotated rx 105.8 ry 33.04 rz -145.95 deg; joints [-6.323, -29.641, 102.77, 144.949, 85.084, 18.944, -295]
  MoveL 2871 to (-3.27, 63.39, -159.35) mm, rotated rx 105.8 ry 33.04 rz -145.95 deg; joints [-6.326, -29.596, 102.734, 144.947, 85.092, 18.939, -295]
  MoveL 2872 to (-2.88, 62.94, -159.37) mm, rotated rx 105.8 ry 33.04 rz -145.95 deg; joints [-6.326, -29.556, 102.702, 144.947, 85.099, 18.934, -295]
  MoveL 2873 to (-2.49, 62.55, -159.38) mm, rotated rx 105.8 ry 33.04 rz -145.95 deg; joints [-6.327, -29.518, 102.67, 144.947, 85.103, 18.932, -295]
  MoveL 2874 to (-2.06, 62.19, -159.38) mm, rotated rx 105.8 ry 33.04 rz -145.95 deg; joints [-6.327, -29.481, 102.634, 144.947, 85.104, 18.931, -295]
  MoveL 2875 to (-1.55, 61.92, -159.38) mm, rotated rx 105.8 ry 33.04 rz -145.95 deg; joints [-6.326, -29.443, 102.589, 144.947, 85.099, 18.935, -295]
  MoveL 2876 to (-0.98, 61.7, -159.38) mm, rotated rx 105.8 ry 33.04 rz -145.95 deg; joints [-6.326, -29.404, 102.539, 144.947, 85.089, 18.941, -295]
  MoveL 2877 to (-2.28, 62.59, -160.34) mm, rotated rx 105.8 ry 33.04 rz -145.95 deg; joints [-6.364, -29.51, 102.648, 144.91, 85.098, 18.948, -295]
  MoveL 2878 to (-1.05, 62.41, -160.76) mm, rotated rx 105.8 ry 33.04 rz -145.95 deg; joints [-6.379, -29.438, 102.533, 144.893, 85.066, 18.977, -295]
  MoveL 2879 to (0.34, 62.11, -161.09) mm, rotated rx 105.8 ry 33.04 rz -145.95 deg; joints [-6.391, -29.353, 102.406, 144.879, 85.033, 19.004, -295]
  MoveL 2880 to (1.89, 61.69, -161.34) mm, rotated rx 105.8 ry 33.04 rz -145.95 deg; joints [-6.4, -29.255, 102.265, 144.869, 84.999, 19.031, -295]
  MoveL 2881 to (3.92, 61.03, -161.45) mm, rotated rx 105.8 ry 33.04 rz -145.95 deg; joints [-6.402, -29.121, 102.081, 144.863, 84.959, 19.06, -295]
  MoveL 2882 to (5.95, 60.38, -161.68) mm, rotated rx 105.8 ry 33.04 rz -145.95 deg; joints [-6.41, -28.988, 101.897, 144.854, 84.918, 19.091, -295]
  MoveL 2883 to (7.97, 59.71, -161.79) mm, rotated rx 105.8 ry 33.04 rz -145.95 deg; joints [-6.413, -28.854, 101.713, 144.848, 84.878, 19.121, -295]
  MoveL 2884 to (10, 59.04, -161.91) mm, rotated rx 105.8 ry 33.04 rz -145.95 deg; joints [-6.416, -28.72, 101.529, 144.843, 84.838, 19.151, -295]
  MoveL 2885 to (12.02, 58.38, -162.14) mm, rotated rx 105.8 ry 33.04 rz -145.95 deg; joints [-6.424, -28.587, 101.344, 144.832, 84.797, 19.182, -295]
  MoveL 2886 to (14.05, 57.7, -162.27) mm, rotated rx 105.8 ry 33.04 rz -145.95 deg; joints [-6.427, -28.453, 101.16, 144.827, 84.756, 19.212, -295]
  MoveL 2887 to (16.07, 57.02, -162.38) mm, rotated rx 105.8 ry 33.04 rz -145.95 deg; joints [-6.43, -28.318, 100.975, 144.821, 84.716, 19.242, -295]
  MoveL 2888 to (18.4, 56.24, -162.54) mm, rotated rx 105.8 ry 33.04 rz -145.95 deg; joints [-6.434, -28.164, 100.761, 144.813, 84.668, 19.277, -295]
  MoveL 2889 to (20.39, 55.57, -162.74) mm, rotated rx 105.8 ry 33.04 rz -145.95 deg; joints [-6.44, -28.031, 100.579, 144.805, 84.628, 19.308, -295]
  MoveL 2890 to (22.58, 54.83, -162.94) mm, rotated rx 105.8 ry 33.04 rz -145.95 deg; joints [-6.446, -27.885, 100.378, 144.796, 84.584, 19.342, -295]
  MoveL 2891 to (24.71, 54.09, -163.19) mm, rotated rx 105.8 ry 33.04 rz -145.95 deg; joints [-6.454, -27.743, 100.18, 144.785, 84.541, 19.375, -295]
  MoveL 2892 to (26.73, 53.4, -163.31) mm, rotated rx 105.8 ry 33.04 rz -145.95 deg; joints [-6.458, -27.608, 99.994, 144.779, 84.5, 19.406, -295]
  MoveL 2893 to (28.75, 52.71, -163.31) mm, rotated rx 105.8 ry 33.04 rz -145.95 deg; joints [-6.456, -27.473, 99.808, 144.777, 84.457, 19.435, -295]
  MoveL 2894 to (30.74, 52.02, -163.39) mm, rotated rx 105.8 ry 33.04 rz -145.95 deg; joints [-6.458, -27.34, 99.624, 144.773, 84.416, 19.465, -295]
  MoveL 2895 to (32.68, 51.33, -163.6) mm, rotated rx 105.8 ry 33.04 rz -145.95 deg; joints [-6.465, -27.209, 99.444, 144.764, 84.377, 19.495, -295]
  MoveL 2896 to (34.84, 50.54, -163.95) mm, rotated rx 105.8 ry 33.04 rz -145.95 deg; joints [-6.476, -27.062, 99.243, 144.749, 84.335, 19.53, -295]
  MoveL 2897 to (36.54, 49.92, -164.16) mm, rotated rx 105.8 ry 33.04 rz -145.95 deg; joints [-6.483, -26.947, 99.085, 144.74, 84.301, 19.556, -295]
  MoveL 2898 to (38.84, 49.05, -164.46) mm, rotated rx 105.8 ry 33.04 rz -145.95 deg; joints [-6.493, -26.79, 98.871, 144.727, 84.256, 19.592, -295]
  MoveL 2899 to (40.92, 48.31, -164.57) mm, rotated rx 105.8 ry 33.04 rz -145.95 deg; joints [-6.496, -26.649, 98.676, 144.721, 84.213, 19.624, -295]
  MoveL 2900 to (42.93, 47.62, -164.58) mm, rotated rx 105.8 ry 33.04 rz -145.95 deg; joints [-6.495, -26.515, 98.488, 144.719, 84.169, 19.655, -295]
  MoveL 2901 to (43.47, 46.91, -165.37) mm, rotated rx 105.8 ry 33.04 rz -145.95 deg; joints [-6.525, -26.456, 98.44, 144.69, 84.183, 19.656, -295]
  MoveL 2902 to (43.03, 46.88, -165.76) mm, rotated rx 105.8 ry 33.04 rz -145.95 deg; joints [-6.54, -26.477, 98.482, 144.677, 84.203, 19.648, -295]
  MoveL 2903 to (42.89, 46.88, -166) mm, rotated rx 105.8 ry 33.04 rz -145.95 deg; joints [-6.55, -26.484, 98.495, 144.668, 84.209, 19.647, -295]
  MoveL 2904 to (43.03, 46.91, -166.13) mm, rotated rx 105.8 ry 33.04 rz -145.95 deg; joints [-6.554, -26.479, 98.481, 144.663, 84.203, 19.653, -295]
  MoveL 2905 to (43.41, 47, -166.15) mm, rotated rx 105.8 ry 33.04 rz -145.95 deg; joints [-6.554, -26.462, 98.442, 144.661, 84.185, 19.666, -295]
  MoveL 2906 to (43.87, 47.11, -166.16) mm, rotated rx 105.8 ry 33.04 rz -145.95 deg; joints [-6.554, -26.443, 98.397, 144.66, 84.164, 19.681, -295]
  MoveL 2907 to (45.38, 47.52, -166.16) mm, rotated rx 105.8 ry 33.04 rz -145.95 deg; joints [-6.552, -26.381, 98.246, 144.657, 84.091, 19.732, -295]
  MoveL 2908 to (45.92, 47.65, -166.18) mm, rotated rx 105.8 ry 33.04 rz -145.95 deg; joints [-6.552, -26.358, 98.192, 144.655, 84.065, 19.75, -295]
  MoveL 2909 to (46.46, 47.77, -166.22) mm, rotated rx 105.8 ry 33.04 rz -145.95 deg; joints [-6.553, -26.334, 98.138, 144.652, 84.041, 19.768, -295]
  MoveL 2910 to (47.03, 47.86, -166.31) mm, rotated rx 105.8 ry 33.04 rz -145.95 deg; joints [-6.556, -26.309, 98.082, 144.648, 84.017, 19.786, -295]
  MoveL 2911 to (47.57, 47.97, -166.37) mm, rotated rx 105.8 ry 33.04 rz -145.95 deg; joints [-6.557, -26.284, 98.028, 144.644, 83.992, 19.804, -295]
  MoveL 2912 to (48.09, 48.09, -166.39) mm, rotated rx 105.8 ry 33.04 rz -145.95 deg; joints [-6.558, -26.262, 97.976, 144.642, 83.968, 19.821, -295]
  MoveL 2913 to (48.57, 48.2, -166.41) mm, rotated rx 105.8 ry 33.04 rz -145.95 deg; joints [-6.558, -26.242, 97.928, 144.64, 83.946, 19.838, -295]
  MoveL 2914 to (49.02, 48.29, -166.45) mm, rotated rx 105.8 ry 33.04 rz -145.95 deg; joints [-6.559, -26.222, 97.883, 144.638, 83.926, 19.852, -295]
  MoveL 2915 to (49.45, 48.38, -166.49) mm, rotated rx 105.8 ry 33.04 rz -145.95 deg; joints [-6.56, -26.202, 97.839, 144.635, 83.906, 19.867, -295]
  MoveL 2916 to (49.94, 48.5, -166.51) mm, rotated rx 105.8 ry 33.04 rz -145.95 deg; joints [-6.56, -26.182, 97.791, 144.634, 83.883, 19.883, -295]
  MoveL 2917 to (50.51, 48.63, -166.53) mm, rotated rx 105.8 ry 33.04 rz -145.95 deg; joints [-6.56, -26.158, 97.734, 144.632, 83.857, 19.902, -295]
  MoveL 2918 to (51.19, 48.77, -166.58) mm, rotated rx 105.8 ry 33.04 rz -145.95 deg; joints [-6.561, -26.127, 97.665, 144.628, 83.825, 19.925, -295]
  MoveL 2919 to (51.78, 48.91, -166.61) mm, rotated rx 105.8 ry 33.04 rz -145.95 deg; joints [-6.561, -26.102, 97.606, 144.626, 83.798, 19.944, -295]
  MoveL 2920 to (53.82, 49.45, -166.61) mm, rotated rx 105.8 ry 33.04 rz -145.95 deg; joints [-6.559, -26.017, 97.401, 144.62, 83.7, 20.014, -295]
  MoveL 2921 to (56.69, 49.93, -166.94) mm, rotated rx 105.8 ry 33.04 rz -145.95 deg; joints [-6.568, -25.885, 97.113, 144.602, 83.575, 20.106, -295]
  MoveL 2922 to (57.98, 49.9, -167.35) mm, rotated rx 105.8 ry 33.04 rz -145.95 deg; joints [-6.582, -25.815, 96.985, 144.584, 83.53, 20.144, -295]
  MoveL 2923 to (59.18, 49.7, -167.93) mm, rotated rx 105.8 ry 33.04 rz -145.95 deg; joints [-6.602, -25.742, 96.867, 144.561, 83.497, 20.176, -295]
  MoveL 2924 to (61.29, 48.77, -169.58) mm, rotated rx 105.8 ry 33.04 rz -145.95 deg; joints [-6.663, -25.59, 96.664, 144.498, 83.466, 20.222, -295]
  MoveL 2925 to (63.02, 47.13, -171.89) mm, rotated rx 105.8 ry 33.04 rz -145.95 deg; joints [-6.749, -25.429, 96.502, 144.414, 83.482, 20.246, -295]
  MoveL 2926 to (63.97, 45.34, -174.19) mm, rotated rx 105.8 ry 33.04 rz -145.95 deg; joints [-6.837, -25.302, 96.418, 144.331, 83.533, 20.244, -295]
  MoveL 2927 to (64, 44.59, -175.1) mm, rotated rx 105.8 ry 33.04 rz -145.95 deg; joints [-6.872, -25.269, 96.418, 144.3, 83.567, 20.233, -295]
  MoveL 2928 to (63.75, 43.94, -175.84) mm, rotated rx 105.8 ry 33.04 rz -145.95 deg; joints [-6.9, -25.255, 96.447, 144.274, 83.608, 20.215, -295]
  MoveL 2929 to (63.51, 43.65, -176.15) mm, rotated rx 105.8 ry 33.04 rz -145.95 deg; joints [-6.913, -25.255, 96.472, 144.264, 83.63, 20.204, -295]
  MoveL 2930 to (63.2, 43.39, -176.42) mm, rotated rx 105.8 ry 33.04 rz -145.95 deg; joints [-6.923, -25.26, 96.505, 144.255, 83.654, 20.191, -295]
  MoveL 2931 to (62.36, 42.93, -176.83) mm, rotated rx 105.8 ry 33.04 rz -145.95 deg; joints [-6.94, -25.286, 96.591, 144.243, 83.707, 20.16, -295]
  MoveL 2932 to (61.22, 42.58, -177.08) mm, rotated rx 105.8 ry 33.04 rz -145.95 deg; joints [-6.952, -25.33, 96.705, 144.236, 83.765, 20.122, -295]
  MoveL 2933 to (59.79, 42.31, -177.16) mm, rotated rx 105.8 ry 33.04 rz -145.95 deg; joints [-6.957, -25.395, 96.848, 144.236, 83.83, 20.077, -295]
  MoveL 2934 to (56.16, 41.83, -177.16) mm, rotated rx 105.8 ry 33.04 rz -145.95 deg; joints [-6.962, -25.566, 97.211, 144.243, 83.986, 19.966, -295]
  MoveL 2935 to (55.7, 41.77, -177.14) mm, rotated rx 105.8 ry 33.04 rz -145.95 deg; joints [-6.962, -25.588, 97.256, 144.244, 84.005, 19.952, -295]
  MoveL 2936 to (55.29, 41.74, -177.12) mm, rotated rx 105.8 ry 33.04 rz -145.95 deg; joints [-6.962, -25.608, 97.297, 144.246, 84.022, 19.94, -295]
  MoveL 2937 to (54.82, 41.69, -177.1) mm, rotated rx 105.8 ry 33.04 rz -145.95 deg; joints [-6.962, -25.631, 97.344, 144.247, 84.041, 19.926, -295]
  MoveL 2938 to (51.19, 41.2, -177.1) mm, rotated rx 105.8 ry 33.04 rz -145.95 deg; joints [-6.967, -25.801, 97.704, 144.254, 84.197, 19.815, -295]
  MoveL 2939 to (50.65, 41.15, -177.08) mm, rotated rx 105.8 ry 33.04 rz -145.95 deg; joints [-6.967, -25.828, 97.758, 144.255, 84.218, 19.8, -295]
  MoveL 2940 to (50.1, 41.13, -177.04) mm, rotated rx 105.8 ry 33.04 rz -145.95 deg; joints [-6.966, -25.855, 97.811, 144.257, 84.239, 19.784, -295]
  MoveL 2941 to (49.62, 41.16, -177) mm, rotated rx 105.8 ry 33.04 rz -145.95 deg; joints [-6.965, -25.882, 97.859, 144.26, 84.256, 19.772, -295]
  MoveL 2942 to (49.24, 41.22, -176.94) mm, rotated rx 105.8 ry 33.04 rz -145.95 deg; joints [-6.963, -25.905, 97.895, 144.262, 84.267, 19.763, -295]
  MoveL 2943 to (49.06, 41.28, -176.77) mm, rotated rx 105.8 ry 33.04 rz -145.95 deg; joints [-6.957, -25.917, 97.913, 144.269, 84.27, 19.758, -295]
  MoveL 2944 to (49.05, 41.32, -176.44) mm, rotated rx 105.8 ry 33.04 rz -145.95 deg; joints [-6.945, -25.919, 97.915, 144.281, 84.268, 19.755, -295]
  MoveL 2945 to (49.2, 41.32, -175.93) mm, rotated rx 105.8 ry 33.04 rz -145.95 deg; joints [-6.925, -25.912, 97.901, 144.3, 84.26, 19.754, -295]
  MoveL 2946 to (48.89, 42.09, -174.47) mm, rotated rx 105.8 ry 33.04 rz -145.95 deg; joints [-6.869, -25.962, 97.929, 144.353, 84.232, 19.753, -295]
  MoveL 2947 to (45.07, 43.97, -174.47) mm, rotated rx 105.8 ry 33.04 rz -145.95 deg; joints [-6.872, -26.242, 98.284, 144.354, 84.293, 19.71, -295]
  MoveL 2948 to (43.24, 44.88, -174.42) mm, rotated rx 105.8 ry 33.04 rz -145.95 deg; joints [-6.872, -26.376, 98.453, 144.357, 84.321, 19.689, -295]
  MoveL 2949 to (41.47, 45.76, -174.33) mm, rotated rx 105.8 ry 33.04 rz -145.95 deg; joints [-6.87, -26.506, 98.617, 144.361, 84.348, 19.669, -295]
  MoveL 2950 to (39.66, 46.65, -174.25) mm, rotated rx 105.8 ry 33.04 rz -145.95 deg; joints [-6.868, -26.639, 98.784, 144.364, 84.375, 19.649, -295]
  MoveL 2951 to (37.89, 47.52, -174.15) mm, rotated rx 105.8 ry 33.04 rz -145.95 deg; joints [-6.866, -26.769, 98.946, 144.369, 84.401, 19.629, -295]
  MoveL 2952 to (36.03, 48.47, -174.11) mm, rotated rx 105.8 ry 33.04 rz -145.95 deg; joints [-6.866, -26.907, 99.117, 144.371, 84.428, 19.61, -295]
  MoveL 2953 to (34.1, 49.54, -174.07) mm, rotated rx 105.8 ry 33.04 rz -145.95 deg; joints [-6.866, -27.053, 99.292, 144.372, 84.452, 19.593, -295]
  MoveL 2954 to (31.82, 50.56, -173.91) mm, rotated rx 105.8 ry 33.04 rz -145.95 deg; joints [-6.861, -27.215, 99.502, 144.379, 84.489, 19.564, -295]
  MoveL 2955 to (29.81, 51.55, -173.66) mm, rotated rx 105.8 ry 33.04 rz -145.95 deg; joints [-6.853, -27.363, 99.686, 144.389, 84.518, 19.54, -295]
  MoveL 2956 to (27.84, 52.52, -173.53) mm, rotated rx 105.8 ry 33.04 rz -145.95 deg; joints [-6.85, -27.507, 99.866, 144.394, 84.546, 19.519, -295]
  MoveL 2957 to (25.92, 53.46, -173.29) mm, rotated rx 105.8 ry 33.04 rz -145.95 deg; joints [-6.842, -27.647, 100.04, 144.404, 84.573, 19.497, -295]
  MoveL 2958 to (24, 54.39, -173.17) mm, rotated rx 105.8 ry 33.04 rz -145.95 deg; joints [-6.839, -27.787, 100.214, 144.409, 84.6, 19.476, -295]
  MoveL 2959 to (22.08, 55.33, -173.05) mm, rotated rx 105.8 ry 33.04 rz -145.95 deg; joints [-6.836, -27.927, 100.388, 144.414, 84.626, 19.456, -295]
  MoveL 2960 to (20.16, 56.25, -172.81) mm, rotated rx 105.8 ry 33.04 rz -145.95 deg; joints [-6.828, -28.067, 100.562, 144.423, 84.653, 19.434, -295]
  MoveL 2961 to (18.24, 57.18, -172.69) mm, rotated rx 105.8 ry 33.04 rz -145.95 deg; joints [-6.825, -28.207, 100.736, 144.428, 84.68, 19.413, -295]
  MoveL 2962 to (16.32, 58.1, -172.57) mm, rotated rx 105.8 ry 33.04 rz -145.95 deg; joints [-6.822, -28.347, 100.909, 144.432, 84.707, 19.393, -295]
  MoveL 2963 to (14.39, 59.03, -172.45) mm, rotated rx 105.8 ry 33.04 rz -145.95 deg; joints [-6.819, -28.486, 101.081, 144.437, 84.733, 19.373, -295]
  MoveL 2964 to (12.46, 59.93, -172.22) mm, rotated rx 105.8 ry 33.04 rz -145.95 deg; joints [-6.812, -28.626, 101.255, 144.446, 84.76, 19.351, -295]
  MoveL 2965 to (10.53, 60.85, -172.11) mm, rotated rx 105.8 ry 33.04 rz -145.95 deg; joints [-6.809, -28.765, 101.428, 144.451, 84.786, 19.331, -295]
  MoveL 2966 to (8.9, 61.58, -171.86) mm, rotated rx 105.8 ry 33.04 rz -145.95 deg; joints [-6.801, -28.882, 101.574, 144.46, 84.809, 19.312, -295]
  MoveL 2967 to (7.39, 62.24, -171.54) mm, rotated rx 105.8 ry 33.04 rz -145.95 deg; joints [-6.789, -28.989, 101.711, 144.473, 84.831, 19.292, -295]
  MoveL 2968 to (5.94, 62.84, -171.12) mm, rotated rx 105.8 ry 33.04 rz -145.95 deg; joints [-6.774, -29.09, 101.843, 144.489, 84.853, 19.271, -295]
  MoveL 2969 to (7.04, 61.5, -170.16) mm, rotated rx 105.8 ry 33.04 rz -145.95 deg; joints [-6.737, -28.976, 101.756, 144.527, 84.87, 19.245, -295]
  MoveL 2970 to (6.5, 61.82, -170.04) mm, rotated rx 105.8 ry 33.04 rz -145.95 deg; joints [-6.733, -29.018, 101.805, 144.532, 84.874, 19.24, -295]
  MoveL 2971 to (6.03, 62.17, -169.95) mm, rotated rx 105.8 ry 33.04 rz -145.95 deg; joints [-6.729, -29.057, 101.845, 144.535, 84.874, 19.239, -295]
  MoveL 2972 to (5.66, 62.57, -169.92) mm, rotated rx 105.8 ry 33.04 rz -145.95 deg; joints [-6.728, -29.093, 101.875, 144.536, 84.869, 19.242, -295]
  MoveL 2973 to (5.35, 63, -169.9) mm, rotated rx 105.8 ry 33.04 rz -145.95 deg; joints [-6.728, -29.128, 101.9, 144.536, 84.861, 19.248, -295]
  MoveL 2974 to (3.48, 66.17, -169.89) mm, rotated rx 105.8 ry 33.04 rz -145.95 deg; joints [-6.726, -29.361, 102.039, 144.532, 84.784, 19.302, -295]
  MoveL 2975 to (3.24, 66.57, -169.88) mm, rotated rx 105.8 ry 33.04 rz -145.95 deg; joints [-6.726, -29.391, 102.057, 144.532, 84.775, 19.309, -295]
  MoveL 2976 to (3.02, 66.92, -169.85) mm, rotated rx 105.8 ry 33.04 rz -145.95 deg; joints [-6.725, -29.418, 102.075, 144.533, 84.766, 19.314, -295]
  MoveL 2977 to (2.77, 67.33, -169.84) mm, rotated rx 105.8 ry 33.04 rz -145.95 deg; joints [-6.724, -29.449, 102.093, 144.532, 84.756, 19.321, -295]
  MoveL 2978 to (2.51, 67.79, -169.84) mm, rotated rx 105.8 ry 33.04 rz -145.95 deg; joints [-6.724, -29.482, 102.113, 144.532, 84.745, 19.329, -295]
  MoveL 2979 to (1.72, 69.15, -169.84) mm, rotated rx 105.8 ry 33.04 rz -145.95 deg; joints [-6.724, -29.581, 102.17, 144.53, 84.711, 19.353, -295]
  MoveL 2980 to (1.4, 69.68, -169.82) mm, rotated rx 105.8 ry 33.04 rz -145.95 deg; joints [-6.723, -29.621, 102.195, 144.53, 84.699, 19.362, -295]
  MoveL 2981 to (1.01, 70.29, -169.78) mm, rotated rx 105.8 ry 33.04 rz -145.95 deg; joints [-6.721, -29.667, 102.224, 144.531, 84.684, 19.372, -295]
  MoveL 2982 to (0.68, 70.84, -169.76) mm, rotated rx 105.8 ry 33.04 rz -145.95 deg; joints [-6.72, -29.708, 102.249, 144.531, 84.671, 19.381, -295]
  MoveL 2983 to (0.15, 71.75, -169.76) mm, rotated rx 105.8 ry 33.04 rz -145.95 deg; joints [-6.72, -29.774, 102.287, 144.529, 84.648, 19.397, -295]
  MoveL 2984 to (-0.51, 73.03, -169.85) mm, rotated rx 105.8 ry 33.04 rz -145.95 deg; joints [-6.723, -29.864, 102.333, 144.524, 84.614, 19.423, -295]
  MoveL 2985 to (-0.91, 74.15, -170.1) mm, rotated rx 105.8 ry 33.04 rz -145.95 deg; joints [-6.732, -29.933, 102.357, 144.513, 84.579, 19.452, -295]
  MoveL 2986 to (-1.06, 75.09, -170.52) mm, rotated rx 105.8 ry 33.04 rz -145.95 deg; joints [-6.748, -29.98, 102.358, 144.495, 84.543, 19.483, -295]
  MoveL 2987 to (-1.03, 75.5, -170.79) mm, rotated rx 105.8 ry 33.04 rz -145.95 deg; joints [-6.758, -29.996, 102.35, 144.484, 84.525, 19.499, -295]
  MoveL 2988 to (-0.94, 75.86, -171.11) mm, rotated rx 105.8 ry 33.04 rz -145.95 deg; joints [-6.77, -30.007, 102.336, 144.471, 84.507, 19.517, -295]
  MoveL 2989 to (-0.57, 76.45, -171.86) mm, rotated rx 105.8 ry 33.04 rz -145.95 deg; joints [-6.798, -30.012, 102.291, 144.44, 84.472, 19.553, -295]
  MoveL 2990 to (0.07, 76.88, -172.79) mm, rotated rx 105.8 ry 33.04 rz -145.95 deg; joints [-6.833, -29.997, 102.223, 144.404, 84.435, 19.592, -295]
  MoveL 2991 to (2.11, 77.2, -175.14) mm, rotated rx 105.8 ry 33.04 rz -145.95 deg; joints [-6.921, -29.902, 102.019, 144.311, 84.363, 19.678, -295]
  MoveL 2992 to (4.51, 76.81, -177.49) mm, rotated rx 105.8 ry 33.04 rz -145.95 deg; joints [-7.009, -29.758, 101.79, 144.22, 84.309, 19.75, -295]
  MoveL 2993 to (6.57, 75.7, -179.17) mm, rotated rx 105.8 ry 33.04 rz -145.95 deg; joints [-7.073, -29.601, 101.604, 144.157, 84.296, 19.784, -295]
  MoveL 2994 to (7.48, 74.87, -179.76) mm, rotated rx 105.8 ry 33.04 rz -145.95 deg; joints [-7.095, -29.518, 101.526, 144.135, 84.305, 19.786, -295]
  MoveL 2995 to (8.3, 73.86, -180.18) mm, rotated rx 105.8 ry 33.04 rz -145.95 deg; joints [-7.111, -29.432, 101.46, 144.12, 84.324, 19.778, -295]
  MoveL 2996 to (9.69, 71.29, -180.51) mm, rotated rx 105.8 ry 33.04 rz -145.95 deg; joints [-7.125, -29.25, 101.358, 144.112, 84.391, 19.734, -295]
  MoveL 2997 to (10.89, 68.39, -180.51) mm, rotated rx 105.8 ry 33.04 rz -145.95 deg; joints [-7.126, -29.063, 101.278, 144.117, 84.478, 19.672, -295]
  MoveL 2998 to (11.32, 67.51, -180.56) mm, rotated rx 105.8 ry 33.04 rz -145.95 deg; joints [-7.128, -29.004, 101.248, 144.116, 84.503, 19.655, -295]
  MoveL 2999 to (11.52, 67.02, -180.56) mm, rotated rx 105.8 ry 33.04 rz -145.95 deg; joints [-7.128, -28.972, 101.235, 144.117, 84.517, 19.644, -295]
  MoveL 3000 to (11.73, 66.52, -180.56) mm, rotated rx 105.8 ry 33.04 rz -145.95 deg; joints [-7.129, -28.94, 101.221, 144.118, 84.532, 19.634, -295]
  MoveL 3001 to (11.96, 66.01, -180.59) mm, rotated rx 105.8 ry 33.04 rz -145.95 deg; joints [-7.13, -28.906, 101.205, 144.118, 84.547, 19.623, -295]
  MoveL 3002 to (12.24, 65.42, -180.65) mm, rotated rx 105.8 ry 33.04 rz -145.95 deg; joints [-7.132, -28.866, 101.184, 144.116, 84.563, 19.613, -295]
  MoveL 3003 to (12.48, 64.9, -180.68) mm, rotated rx 105.8 ry 33.04 rz -145.95 deg; joints [-7.134, -28.831, 101.167, 144.116, 84.578, 19.602, -295]
  MoveL 3004 to (12.69, 64.42, -180.69) mm, rotated rx 105.8 ry 33.04 rz -145.95 deg; joints [-7.134, -28.8, 101.153, 144.116, 84.592, 19.593, -295]
  MoveL 3005 to (12.9, 63.98, -180.72) mm, rotated rx 105.8 ry 33.04 rz -145.95 deg; joints [-7.136, -28.771, 101.138, 144.116, 84.604, 19.584, -295]
  MoveL 3006 to (13.1, 63.58, -180.77) mm, rotated rx 105.8 ry 33.04 rz -145.95 deg; joints [-7.138, -28.743, 101.123, 144.114, 84.615, 19.577, -295]
  MoveL 3007 to (13.31, 63.17, -180.81) mm, rotated rx 105.8 ry 33.04 rz -145.95 deg; joints [-7.139, -28.714, 101.108, 144.114, 84.626, 19.57, -295]
  MoveL 3008 to (13.51, 62.7, -180.82) mm, rotated rx 105.8 ry 33.04 rz -145.95 deg; joints [-7.14, -28.684, 101.094, 144.114, 84.639, 19.56, -295]
  MoveL 3009 to (13.72, 62.23, -180.83) mm, rotated rx 105.8 ry 33.04 rz -145.95 deg; joints [-7.14, -28.653, 101.079, 144.114, 84.652, 19.551, -295]
  MoveL 3010 to (13.95, 61.77, -180.83) mm, rotated rx 105.8 ry 33.04 rz -145.95 deg; joints [-7.141, -28.621, 101.063, 144.115, 84.665, 19.542, -295]
  MoveL 3011 to (14.22, 61.36, -180.85) mm, rotated rx 105.8 ry 33.04 rz -145.95 deg; joints [-7.142, -28.589, 101.042, 144.115, 84.674, 19.536, -295]
  MoveL 3012 to (14.52, 60.99, -180.88) mm, rotated rx 105.8 ry 33.04 rz -145.95 deg; joints [-7.143, -28.558, 101.017, 144.114, 84.679, 19.532, -295]
  MoveL 3013 to (14.86, 60.69, -180.93) mm, rotated rx 105.8 ry 33.04 rz -145.95 deg; joints [-7.144, -28.527, 100.988, 144.112, 84.681, 19.532, -295]
  MoveL 3014 to (15.22, 60.41, -180.97) mm, rotated rx 105.8 ry 33.04 rz -145.95 deg; joints [-7.146, -28.496, 100.957, 144.111, 84.681, 19.532, -295]
  MoveL 3015 to (14.19, 61.53, -181.94) mm, rotated rx 105.8 ry 33.04 rz -145.95 deg; joints [-7.183, -28.597, 101.038, 144.073, 84.672, 19.553, -295]
  MoveL 3016 to (15.71, 60.73, -182.32) mm, rotated rx 105.8 ry 33.04 rz -145.95 deg; joints [-7.197, -28.483, 100.901, 144.059, 84.655, 19.57, -295]
  MoveL 3017 to (17.29, 59.83, -182.6) mm, rotated rx 105.8 ry 33.04 rz -145.95 deg; joints [-7.206, -28.363, 100.761, 144.049, 84.641, 19.584, -295]
  MoveL 3018 to (18.95, 58.82, -182.8) mm, rotated rx 105.8 ry 33.04 rz -145.95 deg; joints [-7.212, -28.233, 100.613, 144.042, 84.628, 19.596, -295]
  MoveL 3019 to (20.76, 57.68, -183.02) mm, rotated rx 105.8 ry 33.04 rz -145.95 deg; joints [-7.219, -28.09, 100.452, 144.034, 84.615, 19.608, -295]
  MoveL 3020 to (22.55, 56.52, -183.14) mm, rotated rx 105.8 ry 33.04 rz -145.95 deg; joints [-7.222, -27.947, 100.294, 144.03, 84.602, 19.618, -295]
  MoveL 3021 to (24.34, 55.36, -183.25) mm, rotated rx 105.8 ry 33.04 rz -145.95 deg; joints [-7.225, -27.804, 100.135, 144.026, 84.59, 19.628, -295]
  MoveL 3022 to (26.14, 54.21, -183.48) mm, rotated rx 105.8 ry 33.04 rz -145.95 deg; joints [-7.233, -27.66, 99.974, 144.018, 84.577, 19.64, -295]
  MoveL 3023 to (27.92, 53.04, -183.6) mm, rotated rx 105.8 ry 33.04 rz -145.95 deg; joints [-7.236, -27.517, 99.814, 144.014, 84.565, 19.651, -295]
  MoveL 3024 to (29.71, 51.87, -183.72) mm, rotated rx 105.8 ry 33.04 rz -145.95 deg; joints [-7.239, -27.374, 99.655, 144.01, 84.552, 19.661, -295]
  MoveL 3025 to (31.5, 50.7, -183.96) mm, rotated rx 105.8 ry 33.04 rz -145.95 deg; joints [-7.247, -27.231, 99.494, 144.002, 84.539, 19.673, -295]
  MoveL 3026 to (33.28, 49.53, -184.08) mm, rotated rx 105.8 ry 33.04 rz -145.95 deg; joints [-7.25, -27.088, 99.334, 143.998, 84.526, 19.684, -295]
  MoveL 3027 to (35.06, 48.35, -184.2) mm, rotated rx 105.8 ry 33.04 rz -145.95 deg; joints [-7.253, -26.944, 99.174, 143.994, 84.513, 19.695, -295]
  MoveL 3028 to (36.74, 47.23, -184.39) mm, rotated rx 105.8 ry 33.04 rz -145.95 deg; joints [-7.259, -26.809, 99.022, 143.987, 84.501, 19.706, -295]
  MoveL 3029 to (38.26, 46.22, -184.6) mm, rotated rx 105.8 ry 33.04 rz -145.95 deg; joints [-7.266, -26.686, 98.884, 143.979, 84.49, 19.716, -295]
  MoveL 3030 to (39.89, 45.13, -184.71) mm, rotated rx 105.8 ry 33.04 rz -145.95 deg; joints [-7.269, -26.554, 98.737, 143.976, 84.478, 19.727, -295]
  MoveL 3031 to (41.75, 44.01, -184.71) mm, rotated rx 105.8 ry 33.04 rz -145.95 deg; joints [-7.267, -26.409, 98.567, 143.976, 84.457, 19.741, -295]
  MoveL 3032 to (44.01, 42.49, -184.8) mm, rotated rx 105.8 ry 33.04 rz -145.95 deg; joints [-7.269, -26.226, 98.362, 143.973, 84.44, 19.754, -295]
  MoveL 3033 to (45.98, 41.02, -185.04) mm, rotated rx 105.8 ry 33.04 rz -145.95 deg; joints [-7.276, -26.06, 98.183, 143.965, 84.43, 19.764, -295]
  MoveL 3034 to (47.67, 39.88, -185.22) mm, rotated rx 105.8 ry 33.04 rz -145.95 deg; joints [-7.282, -25.923, 98.029, 143.958, 84.418, 19.775, -295]
  MoveL 3035 to (49.2, 38.81, -185.54) mm, rotated rx 105.8 ry 33.04 rz -145.95 deg; joints [-7.293, -25.797, 97.887, 143.947, 84.407, 19.787, -295]
  MoveL 3036 to (50.89, 37.65, -185.72) mm, rotated rx 105.8 ry 33.04 rz -145.95 deg; joints [-7.298, -25.66, 97.732, 143.94, 84.394, 19.799, -295]
  MoveL 3037 to (52.51, 36.52, -185.92) mm, rotated rx 105.8 ry 33.04 rz -145.95 deg; joints [-7.305, -25.527, 97.584, 143.933, 84.383, 19.81, -295]
  MoveL 3038 to (54.07, 35.4, -186.2) mm, rotated rx 105.8 ry 33.04 rz -145.95 deg; joints [-7.314, -25.397, 97.439, 143.923, 84.373, 19.82, -295]
  MoveL 3039 to (54.37, 34.54, -186.97) mm, rotated rx 105.8 ry 33.04 rz -145.95 deg; joints [-7.344, -25.344, 97.414, 143.896, 84.401, 19.811, -295]
  MoveL 3040 to (54, 34.56, -187.35) mm, rotated rx 105.8 ry 33.04 rz -145.95 deg; joints [-7.359, -25.364, 97.449, 143.882, 84.415, 19.807, -295]
  MoveL 3041 to (53.92, 34.54, -187.59) mm, rotated rx 105.8 ry 33.04 rz -145.95 deg; joints [-7.368, -25.367, 97.456, 143.873, 84.42, 19.806, -295]
  MoveL 3042 to (54.12, 34.48, -187.72) mm, rotated rx 105.8 ry 33.04 rz -145.95 deg; joints [-7.373, -25.354, 97.436, 143.868, 84.415, 19.812, -295]
  MoveL 3043 to (54.65, 34.43, -187.77) mm, rotated rx 105.8 ry 33.04 rz -145.95 deg; joints [-7.374, -25.324, 97.385, 143.866, 84.399, 19.824, -295]
  MoveL 3044 to (55.31, 34.38, -187.81) mm, rotated rx 105.8 ry 33.04 rz -145.95 deg; joints [-7.374, -25.287, 97.32, 143.864, 84.376, 19.841, -295]
  MoveL 3045 to (56.88, 34.39, -187.81) mm, rotated rx 105.8 ry 33.04 rz -145.95 deg; joints [-7.372, -25.205, 97.165, 143.862, 84.317, 19.884, -295]
  MoveL 3046 to (57.43, 34.39, -187.81) mm, rotated rx 105.8 ry 33.04 rz -145.95 deg; joints [-7.371, -25.176, 97.111, 143.861, 84.297, 19.898, -295]
  MoveL 3047 to (57.97, 34.37, -187.84) mm, rotated rx 105.8 ry 33.04 rz -145.95 deg; joints [-7.371, -25.147, 97.059, 143.86, 84.277, 19.913, -295]
  MoveL 3048 to (58.52, 34.34, -187.89) mm, rotated rx 105.8 ry 33.04 rz -145.95 deg; joints [-7.372, -25.117, 97.005, 143.857, 84.258, 19.927, -295]
  MoveL 3049 to (59.07, 34.29, -187.96) mm, rotated rx 105.8 ry 33.04 rz -145.95 deg; joints [-7.374, -25.086, 96.95, 143.854, 84.24, 19.941, -295]
  MoveL 3050 to (59.62, 34.25, -188.02) mm, rotated rx 105.8 ry 33.04 rz -145.95 deg; joints [-7.376, -25.055, 96.896, 143.851, 84.221, 19.955, -295]
  MoveL 3051 to (60.12, 34.24, -188.04) mm, rotated rx 105.8 ry 33.04 rz -145.95 deg; joints [-7.376, -25.028, 96.847, 143.85, 84.203, 19.969, -295]
  MoveL 3052 to (60.58, 34.23, -188.06) mm, rotated rx 105.8 ry 33.04 rz -145.95 deg; joints [-7.376, -25.004, 96.802, 143.849, 84.186, 19.981, -295]
  MoveL 3053 to (62.15, 34.24, -188.06) mm, rotated rx 105.8 ry 33.04 rz -145.95 deg; joints [-7.373, -24.922, 96.647, 143.847, 84.127, 20.023, -295]
  MoveL 3054 to (62.67, 34.23, -188.07) mm, rotated rx 105.8 ry 33.04 rz -145.95 deg; joints [-7.373, -24.894, 96.595, 143.845, 84.108, 20.037, -295]
  MoveL 3055 to (63.14, 34.21, -188.1) mm, rotated rx 105.8 ry 33.04 rz -145.95 deg; joints [-7.373, -24.868, 96.548, 143.844, 84.091, 20.05, -295]
  MoveL 3056 to (63.59, 34.18, -188.15) mm, rotated rx 105.8 ry 33.04 rz -145.95 deg; joints [-7.375, -24.843, 96.505, 143.842, 84.076, 20.061, -295]
  MoveL 3057 to (64.04, 34.15, -188.19) mm, rotated rx 105.8 ry 33.04 rz -145.95 deg; joints [-7.375, -24.818, 96.46, 143.84, 84.06, 20.073, -295]
  MoveL 3058 to (64.53, 34.14, -188.2) mm, rotated rx 105.8 ry 33.04 rz -145.95 deg; joints [-7.375, -24.792, 96.411, 143.838, 84.042, 20.087, -295]
  MoveL 3059 to (65.05, 34.15, -188.2) mm, rotated rx 105.8 ry 33.04 rz -145.95 deg; joints [-7.374, -24.764, 96.359, 143.838, 84.022, 20.101, -295]
  MoveL 3060 to (67.97, 33.87, -188.54) mm, rotated rx 105.8 ry 33.04 rz -145.95 deg; joints [-7.383, -24.598, 96.071, 143.822, 83.926, 20.175, -295]
  MoveL 3061 to (69.23, 33.5, -188.96) mm, rotated rx 105.8 ry 33.04 rz -145.95 deg; joints [-7.397, -24.515, 95.947, 143.805, 83.894, 20.204, -295]
  MoveL 3062 to (70.37, 33, -189.55) mm, rotated rx 105.8 ry 33.04 rz -145.95 deg; joints [-7.418, -24.433, 95.836, 143.783, 83.875, 20.227, -295]
  MoveL 3063 to (72.26, 31.53, -191.24) mm, rotated rx 105.8 ry 33.04 rz -145.95 deg; joints [-7.48, -24.27, 95.653, 143.721, 83.871, 20.254, -295]
  MoveL 3064 to (73.62, 29.48, -193.6) mm, rotated rx 105.8 ry 33.04 rz -145.95 deg; joints [-7.569, -24.109, 95.523, 143.637, 83.913, 20.259, -295]
  MoveL 3065 to (74.2, 27.48, -195.96) mm, rotated rx 105.8 ry 33.04 rz -145.95 deg; joints [-7.659, -23.992, 95.471, 143.553, 83.982, 20.243, -295]
  MoveL 3066 to (74.09, 26.73, -196.89) mm, rotated rx 105.8 ry 33.04 rz -145.95 deg; joints [-7.694, -23.965, 95.484, 143.521, 84.021, 20.229, -295]
  MoveL 3067 to (73.71, 26.16, -197.65) mm, rotated rx 105.8 ry 33.04 rz -145.95 deg; joints [-7.724, -23.96, 95.522, 143.494, 84.061, 20.21, -295]
  MoveL 3068 to (73.43, 25.94, -197.97) mm, rotated rx 105.8 ry 33.04 rz -145.95 deg; joints [-7.737, -23.966, 95.551, 143.483, 84.083, 20.199, -295]
  MoveL 3069 to (73.07, 25.76, -198.24) mm, rotated rx 105.8 ry 33.04 rz -145.95 deg; joints [-7.748, -23.976, 95.587, 143.474, 84.105, 20.187, -295]
  MoveL 3070 to (72.16, 25.53, -198.66) mm, rotated rx 105.8 ry 33.04 rz -145.95 deg; joints [-7.766, -24.014, 95.677, 143.46, 84.15, 20.16, -295]
  MoveL 3071 to (70.98, 25.47, -198.92) mm, rotated rx 105.8 ry 33.04 rz -145.95 deg; joints [-7.778, -24.073, 95.794, 143.452, 84.199, 20.129, -295]
  MoveL 3072 to (69.54, 25.58, -199) mm, rotated rx 105.8 ry 33.04 rz -145.95 deg; joints [-7.783, -24.154, 95.936, 143.45, 84.249, 20.093, -295]
  MoveL 3073 to (67.98, 25.77, -199) mm, rotated rx 105.8 ry 33.04 rz -145.95 deg; joints [-7.786, -24.244, 96.089, 143.451, 84.3, 20.056, -295]
  MoveL 3074 to (67.46, 25.84, -199) mm, rotated rx 105.8 ry 33.04 rz -145.95 deg; joints [-7.786, -24.275, 96.141, 143.452, 84.317, 20.044, -295]
  MoveL 3075 to (66.89, 25.93, -198.96) mm, rotated rx 105.8 ry 33.04 rz -145.95 deg; joints [-7.786, -24.309, 96.197, 143.454, 84.335, 20.031, -295]
  MoveL 3076 to (66.26, 26.06, -198.9) mm, rotated rx 105.8 ry 33.04 rz -145.95 deg; joints [-7.785, -24.347, 96.259, 143.456, 84.353, 20.016, -295]
  MoveL 3077 to (65.7, 26.15, -198.87) mm, rotated rx 105.8 ry 33.04 rz -145.95 deg; joints [-7.785, -24.38, 96.313, 143.458, 84.371, 20.004, -295]
  MoveL 3078 to (65.18, 26.22, -198.87) mm, rotated rx 105.8 ry 33.04 rz -145.95 deg; joints [-7.785, -24.411, 96.365, 143.458, 84.388, 19.991, -295]
  MoveL 3079 to (64.66, 26.29, -198.86) mm, rotated rx 105.8 ry 33.04 rz -145.95 deg; joints [-7.786, -24.441, 96.415, 143.459, 84.404, 19.979, -295]
  MoveL 3080 to (64.16, 26.38, -198.81) mm, rotated rx 105.8 ry 33.04 rz -145.95 deg; joints [-7.785, -24.471, 96.464, 143.461, 84.419, 19.968, -295]
  MoveL 3081 to (63.67, 26.5, -198.73) mm, rotated rx 105.8 ry 33.04 rz -145.95 deg; joints [-7.783, -24.502, 96.512, 143.464, 84.432, 19.957, -295]
  MoveL 3082 to (63.18, 26.63, -198.64) mm, rotated rx 105.8 ry 33.04 rz -145.95 deg; joints [-7.78, -24.533, 96.56, 143.468, 84.445, 19.946, -295]
  MoveL 3083 to (62.68, 26.74, -198.57) mm, rotated rx 105.8 ry 33.04 rz -145.95 deg; joints [-7.778, -24.564, 96.609, 143.471, 84.459, 19.935, -295]
  MoveL 3084 to (62.16, 26.82, -198.54) mm, rotated rx 105.8 ry 33.04 rz -145.95 deg; joints [-7.778, -24.595, 96.66, 143.472, 84.475, 19.923, -295]
  MoveL 3085 to (61.65, 26.89, -198.53) mm, rotated rx 105.8 ry 33.04 rz -145.95 deg; joints [-7.778, -24.625, 96.71, 143.473, 84.492, 19.911, -295]
  MoveL 3086 to (59.11, 27.25, -198.52) mm, rotated rx 105.8 ry 33.04 rz -145.95 deg; joints [-7.782, -24.773, 96.957, 143.475, 84.572, 19.853, -295]
  MoveL 3087 to (58.74, 27.36, -198.5) mm, rotated rx 105.8 ry 33.04 rz -145.95 deg; joints [-7.782, -24.797, 96.993, 143.476, 84.581, 19.845, -295]
  MoveL 3088 to (58.59, 27.43, -198.38) mm, rotated rx 105.8 ry 33.04 rz -145.95 deg; joints [-7.777, -24.808, 97.008, 143.48, 84.584, 19.842, -295]
  MoveL 3089 to (58.68, 27.41, -198.15) mm, rotated rx 105.8 ry 33.04 rz -145.95 deg; joints [-7.769, -24.803, 97.001, 143.489, 84.581, 19.841, -295]
  MoveL 3090 to (59.01, 27.27, -197.79) mm, rotated rx 105.8 ry 33.04 rz -145.95 deg; joints [-7.754, -24.78, 96.971, 143.502, 84.572, 19.842, -295]
  MoveL 3091 to (58.8, 28.01, -197.05) mm, rotated rx 105.8 ry 33.04 rz -145.95 deg; joints [-7.726, -24.824, 96.989, 143.528, 84.547, 19.85, -295]
  MoveL 3092 to (57.2, 29.4, -197.03) mm, rotated rx 105.8 ry 33.04 rz -145.95 deg; joints [-7.726, -24.967, 97.135, 143.528, 84.549, 19.848, -295]
  MoveL 3093 to (55.57, 30.86, -196.9) mm, rotated rx 105.8 ry 33.04 rz -145.95 deg; joints [-7.723, -25.114, 97.283, 143.532, 84.549, 19.847, -295]
  MoveL 3094 to (53.9, 32.4, -196.64) mm, rotated rx 105.8 ry 33.04 rz -145.95 deg; joints [-7.714, -25.268, 97.435, 143.54, 84.546, 19.846, -295]
  MoveL 3095 to (52.32, 33.82, -196.51) mm, rotated rx 105.8 ry 33.04 rz -145.95 deg; joints [-7.71, -25.41, 97.578, 143.544, 84.545, 19.845, -295]
  MoveL 3096 to (50.81, 35.19, -196.25) mm, rotated rx 105.8 ry 33.04 rz -145.95 deg; joints [-7.701, -25.549, 97.715, 143.553, 84.543, 19.843, -295]
  MoveL 3097 to (49.25, 36.61, -195.89) mm, rotated rx 105.8 ry 33.04 rz -145.95 deg; joints [-7.689, -25.691, 97.856, 143.565, 84.54, 19.841, -295]
  MoveL 3098 to (47.64, 38.03, -195.75) mm, rotated rx 105.8 ry 33.04 rz -145.95 deg; joints [-7.685, -25.836, 98.001, 143.569, 84.539, 19.84, -295]
  MoveL 3099 to (46.05, 39.42, -195.65) mm, rotated rx 105.8 ry 33.04 rz -145.95 deg; joints [-7.682, -25.978, 98.144, 143.571, 84.539, 19.839, -295]
  MoveL 3100 to (44.43, 40.84, -195.51) mm, rotated rx 105.8 ry 33.04 rz -145.95 deg; joints [-7.678, -26.123, 98.288, 143.575, 84.538, 19.838, -295]
  MoveL 3101 to (42.88, 42.24, -195.22) mm, rotated rx 105.8 ry 33.04 rz -145.95 deg; joints [-7.668, -26.264, 98.427, 143.585, 84.534, 19.837, -295]
  MoveL 3102 to (41.21, 43.64, -194.88) mm, rotated rx 105.8 ry 33.04 rz -145.95 deg; joints [-7.656, -26.412, 98.578, 143.596, 84.534, 19.832, -295]
  MoveL 3103 to (39.6, 45.03, -194.7) mm, rotated rx 105.8 ry 33.04 rz -145.95 deg; joints [-7.65, -26.555, 98.721, 143.602, 84.534, 19.831, -295]
  MoveL 3104 to (37.97, 46.42, -194.59) mm, rotated rx 105.8 ry 33.04 rz -145.95 deg; joints [-7.648, -26.7, 98.865, 143.605, 84.533, 19.83, -295]
  MoveL 3105 to (36.36, 47.81, -194.52) mm, rotated rx 105.8 ry 33.04 rz -145.95 deg; joints [-7.646, -26.843, 99.007, 143.606, 84.531, 19.831, -295]
  MoveL 3106 to (34.73, 49.19, -194.29) mm, rotated rx 105.8 ry 33.04 rz -145.95 deg; joints [-7.639, -26.988, 99.153, 143.614, 84.53, 19.829, -295]
  MoveL 3107 to (33.11, 50.57, -194.16) mm, rotated rx 105.8 ry 33.04 rz -145.95 deg; joints [-7.635, -27.131, 99.295, 143.617, 84.529, 19.828, -295]
  MoveL 3108 to (31.48, 51.97, -194.08) mm, rotated rx 105.8 ry 33.04 rz -145.95 deg; joints [-7.633, -27.275, 99.438, 143.619, 84.527, 19.829, -295]
  MoveL 3109 to (29.85, 53.32, -193.85) mm, rotated rx 105.8 ry 33.04 rz -145.95 deg; joints [-7.625, -27.419, 99.582, 143.626, 84.526, 19.827, -295]
  MoveL 3110 to (28.19, 54.69, -193.62) mm, rotated rx 105.8 ry 33.04 rz -145.95 deg; joints [-7.618, -27.564, 99.728, 143.634, 84.526, 19.824, -295]
  MoveL 3111 to (26.52, 56.09, -193.47) mm, rotated rx 105.8 ry 33.04 rz -145.95 deg; joints [-7.613, -27.711, 99.874, 143.638, 84.524, 19.824, -295]
  MoveL 3112 to (25.06, 57.27, -193.34) mm, rotated rx 105.8 ry 33.04 rz -145.95 deg; joints [-7.61, -27.838, 100.001, 143.642, 84.524, 19.822, -295]
  MoveL 3113 to (23.75, 58.26, -193.13) mm, rotated rx 105.8 ry 33.04 rz -145.95 deg; joints [-7.603, -27.949, 100.117, 143.649, 84.527, 19.818, -295]
  MoveL 3114 to (22.55, 59.06, -192.81) mm, rotated rx 105.8 ry 33.04 rz -145.95 deg; joints [-7.592, -28.046, 100.224, 143.66, 84.533, 19.809, -295]
  MoveL 3115 to (23.51, 57.94, -191.85) mm, rotated rx 105.8 ry 33.04 rz -145.95 deg; joints [-7.554, -27.949, 100.149, 143.698, 84.544, 19.787, -295]
  MoveL 3116 to (23.13, 58.26, -191.85) mm, rotated rx 105.8 ry 33.04 rz -145.95 deg; joints [-7.555, -27.982, 100.182, 143.697, 84.543, 19.787, -295]
  MoveL 3117 to (22.78, 58.62, -191.85) mm, rotated rx 105.8 ry 33.04 rz -145.95 deg; joints [-7.555, -28.016, 100.211, 143.697, 84.54, 19.79, -295]
  MoveL 3118 to (22.49, 59.06, -191.82) mm, rotated rx 105.8 ry 33.04 rz -145.95 deg; joints [-7.554, -28.05, 100.235, 143.698, 84.531, 19.796, -295]
  MoveL 3119 to (22.23, 59.56, -191.78) mm, rotated rx 105.8 ry 33.04 rz -145.95 deg; joints [-7.552, -28.085, 100.254, 143.698, 84.519, 19.804, -295]
  MoveL 3120 to (21.99, 60.12, -191.73) mm, rotated rx 105.8 ry 33.04 rz -145.95 deg; joints [-7.55, -28.121, 100.271, 143.7, 84.502, 19.816, -295]
  MoveL 3121 to (21.81, 60.67, -191.69) mm, rotated rx 105.8 ry 33.04 rz -145.95 deg; joints [-7.548, -28.154, 100.282, 143.7, 84.485, 19.828, -295]
  MoveL 3122 to (21.65, 61.21, -191.67) mm, rotated rx 105.8 ry 33.04 rz -145.95 deg; joints [-7.547, -28.185, 100.292, 143.7, 84.467, 19.841, -295]
  MoveL 3123 to (21.51, 61.72, -191.67) mm, rotated rx 105.8 ry 33.04 rz -145.95 deg; joints [-7.546, -28.214, 100.299, 143.699, 84.449, 19.853, -295]
  MoveL 3124 to (21.37, 62.23, -191.67) mm, rotated rx 105.8 ry 33.04 rz -145.95 deg; joints [-7.546, -28.243, 100.307, 143.698, 84.432, 19.866, -295]
  MoveL 3125 to (21.18, 62.78, -191.62) mm, rotated rx 105.8 ry 33.04 rz -145.95 deg; joints [-7.544, -28.277, 100.319, 143.699, 84.414, 19.878, -295]
  MoveL 3126 to (20.95, 63.4, -191.54) mm, rotated rx 105.8 ry 33.04 rz -145.95 deg; joints [-7.54, -28.315, 100.335, 143.701, 84.395, 19.891, -295]
  MoveL 3127 to (20.78, 63.89, -191.49) mm, rotated rx 105.8 ry 33.04 rz -145.95 deg; joints [-7.538, -28.345, 100.345, 143.702, 84.38, 19.902, -295]
  MoveL 3128 to (20.66, 64.29, -191.46) mm, rotated rx 105.8 ry 33.04 rz -145.95 deg; joints [-7.537, -28.368, 100.353, 143.702, 84.366, 19.911, -295]
  MoveL 3129 to (20.52, 64.76, -191.45) mm, rotated rx 105.8 ry 33.04 rz -145.95 deg; joints [-7.536, -28.395, 100.36, 143.702, 84.351, 19.922, -295]
  MoveL 3130 to (20.38, 65.26, -191.45) mm, rotated rx 105.8 ry 33.04 rz -145.95 deg; joints [-7.536, -28.424, 100.368, 143.701, 84.334, 19.934, -295]
  MoveL 3131 to (20.24, 65.75, -191.43) mm, rotated rx 105.8 ry 33.04 rz -145.95 deg; joints [-7.535, -28.452, 100.376, 143.701, 84.317, 19.946, -295]
  MoveL 3132 to (20.09, 66.22, -191.41) mm, rotated rx 105.8 ry 33.04 rz -145.95 deg; joints [-7.533, -28.48, 100.385, 143.701, 84.302, 19.957, -295]
  MoveL 3133 to (19.95, 66.72, -191.4) mm, rotated rx 105.8 ry 33.04 rz -145.95 deg; joints [-7.533, -28.508, 100.393, 143.701, 84.285, 19.969, -295]
  MoveL 3134 to (19.26, 69.25, -191.39) mm, rotated rx 105.8 ry 33.04 rz -145.95 deg; joints [-7.531, -28.651, 100.429, 143.696, 84.199, 20.032, -295]
  MoveL 3135 to (18.94, 70.67, -191.48) mm, rotated rx 105.8 ry 33.04 rz -145.95 deg; joints [-7.533, -28.728, 100.442, 143.69, 84.148, 20.07, -295]
  MoveL 3136 to (18.82, 71.86, -191.73) mm, rotated rx 105.8 ry 33.04 rz -145.95 deg; joints [-7.541, -28.784, 100.439, 143.678, 84.101, 20.108, -295]
  MoveL 3137 to (18.89, 72.83, -192.14) mm, rotated rx 105.8 ry 33.04 rz -145.95 deg; joints [-7.556, -28.821, 100.418, 143.66, 84.058, 20.146, -295]
  MoveL 3138 to (19.16, 73.57, -192.73) mm, rotated rx 105.8 ry 33.04 rz -145.95 deg; joints [-7.577, -28.837, 100.381, 143.637, 84.019, 20.183, -295]
  MoveL 3139 to (19.63, 74.08, -193.48) mm, rotated rx 105.8 ry 33.04 rz -145.95 deg; joints [-7.605, -28.833, 100.327, 143.607, 83.984, 20.22, -295]
  MoveL 3140 to (20.29, 74.37, -194.39) mm, rotated rx 105.8 ry 33.04 rz -145.95 deg; joints [-7.638, -28.809, 100.256, 143.571, 83.953, 20.257, -295]
  MoveL 3141 to (22.2, 74.26, -196.72) mm, rotated rx 105.8 ry 33.04 rz -145.95 deg; joints [-7.724, -28.701, 100.064, 143.482, 83.901, 20.329, -295]
  MoveL 3142 to (24.3, 73.39, -199.07) mm, rotated rx 105.8 ry 33.04 rz -145.95 deg; joints [-7.811, -28.55, 99.862, 143.394, 83.877, 20.382, -295]
  MoveL 3143 to (25.99, 71.87, -200.77) mm, rotated rx 105.8 ry 33.04 rz -145.95 deg; joints [-7.875, -28.396, 99.71, 143.332, 83.891, 20.397, -295]
  MoveL 3144 to (26.69, 70.88, -201.39) mm, rotated rx 105.8 ry 33.04 rz -145.95 deg; joints [-7.898, -28.317, 99.652, 143.31, 83.913, 20.391, -295]
  MoveL 3145 to (27.28, 69.72, -201.84) mm, rotated rx 105.8 ry 33.04 rz -145.95 deg; joints [-7.916, -28.237, 99.607, 143.295, 83.944, 20.374, -295]
  MoveL 3146 to (28.14, 66.94, -202.27) mm, rotated rx 105.8 ry 33.04 rz -145.95 deg; joints [-7.934, -28.074, 99.554, 143.285, 84.035, 20.313, -295]
  MoveL 3147 to (28.36, 65.95, -202.31) mm, rotated rx 105.8 ry 33.04 rz -145.95 deg; joints [-7.936, -28.021, 99.545, 143.285, 84.071, 20.287, -295]
  MoveL 3148 to (28.72, 63.36, -202.31) mm, rotated rx 105.8 ry 33.04 rz -145.95 deg; joints [-7.939, -27.893, 99.54, 143.29, 84.17, 20.214, -295]
  MoveL 3149 to (28.9, 62.37, -202.37) mm, rotated rx 105.8 ry 33.04 rz -145.95 deg; joints [-7.942, -27.842, 99.533, 143.29, 84.206, 20.188, -295]
  MoveL 3150 to (29.04, 61.33, -202.37) mm, rotated rx 105.8 ry 33.04 rz -145.95 deg; joints [-7.943, -27.79, 99.531, 143.292, 84.246, 20.159, -295]
  MoveL 3151 to (29.12, 60.85, -202.38) mm, rotated rx 105.8 ry 33.04 rz -145.95 deg; joints [-7.944, -27.766, 99.529, 143.292, 84.264, 20.146, -295]
  MoveL 3152 to (29.19, 60.43, -202.4) mm, rotated rx 105.8 ry 33.04 rz -145.95 deg; joints [-7.945, -27.744, 99.526, 143.292, 84.279, 20.135, -295]
  MoveL 3153 to (29.27, 59.97, -202.41) mm, rotated rx 105.8 ry 33.04 rz -145.95 deg; joints [-7.946, -27.721, 99.524, 143.293, 84.296, 20.122, -295]
  MoveL 3154 to (29.63, 57.38, -202.42) mm, rotated rx 105.8 ry 33.04 rz -145.95 deg; joints [-7.949, -27.592, 99.517, 143.297, 84.394, 20.05, -295]
  MoveL 3155 to (29.72, 56.89, -202.44) mm, rotated rx 105.8 ry 33.04 rz -145.95 deg; joints [-7.95, -27.567, 99.514, 143.297, 84.412, 20.036, -295]
  MoveL 3156 to (29.82, 56.44, -202.47) mm, rotated rx 105.8 ry 33.04 rz -145.95 deg; joints [-7.952, -27.542, 99.509, 143.297, 84.428, 20.025, -295]
  MoveL 3157 to (29.95, 56.02, -202.51) mm, rotated rx 105.8 ry 33.04 rz -145.95 deg; joints [-7.954, -27.518, 99.501, 143.296, 84.442, 20.016, -295]
  MoveL 3158 to (30.11, 55.62, -202.55) mm, rotated rx 105.8 ry 33.04 rz -145.95 deg; joints [-7.955, -27.492, 99.489, 143.295, 84.453, 20.008, -295]
  MoveL 3159 to (30.33, 55.24, -202.56) mm, rotated rx 105.8 ry 33.04 rz -145.95 deg; joints [-7.956, -27.465, 99.472, 143.295, 84.462, 20.002, -295]
  MoveL 3160 to (30.59, 54.88, -202.57) mm, rotated rx 105.8 ry 33.04 rz -145.95 deg; joints [-7.956, -27.436, 99.451, 143.296, 84.468, 19.997, -295]
  MoveL 3161 to (30.26, 55.56, -203.31) mm, rotated rx 105.8 ry 33.04 rz -145.95 deg; joints [-7.984, -27.481, 99.471, 143.267, 84.453, 20.019, -295]
  MoveL 3162 to (31.39, 54.67, -203.86) mm, rotated rx 105.8 ry 33.04 rz -145.95 deg; joints [-8.004, -27.384, 99.369, 143.247, 84.453, 20.027, -295]
  MoveL 3163 to (32.55, 53.64, -204.28) mm, rotated rx 105.8 ry 33.04 rz -145.95 deg; joints [-8.019, -27.278, 99.266, 143.232, 84.458, 20.029, -295]
  MoveL 3164 to (33.82, 52.4, -204.59) mm, rotated rx 105.8 ry 33.04 rz -145.95 deg; joints [-8.03, -27.159, 99.156, 143.222, 84.467, 20.027, -295]
  MoveL 3165 to (35.2, 50.93, -204.78) mm, rotated rx 105.8 ry 33.04 rz -145.95 deg; joints [-8.036, -27.024, 99.037, 143.217, 84.481, 20.018, -295]
  MoveL 3166 to (36.63, 49.39, -204.97) mm, rotated rx 105.8 ry 33.04 rz -145.95 deg; joints [-8.043, -26.884, 98.913, 143.212, 84.496, 20.01, -295]
  MoveL 3167 to (38.06, 47.81, -205.09) mm, rotated rx 105.8 ry 33.04 rz -145.95 deg; joints [-8.046, -26.741, 98.79, 143.209, 84.512, 19.999, -295]
  MoveL 3168 to (39.5, 46.24, -205.32) mm, rotated rx 105.8 ry 33.04 rz -145.95 deg; joints [-8.054, -26.599, 98.665, 143.203, 84.527, 19.991, -295]
  MoveL 3169 to (40.93, 44.65, -205.43) mm, rotated rx 105.8 ry 33.04 rz -145.95 deg; joints [-8.058, -26.456, 98.541, 143.2, 84.543, 19.981, -295]
  MoveL 3170 to (42.36, 43.07, -205.55) mm, rotated rx 105.8 ry 33.04 rz -145.95 deg; joints [-8.061, -26.314, 98.417, 143.198, 84.558, 19.97, -295]
  MoveL 3171 to (43.79, 41.48, -205.66) mm, rotated rx 105.8 ry 33.04 rz -145.95 deg; joints [-8.065, -26.172, 98.293, 143.195, 84.573, 19.96, -295]
  MoveL 3172 to (45.22, 39.9, -205.9) mm, rotated rx 105.8 ry 33.04 rz -145.95 deg; joints [-8.073, -26.029, 98.168, 143.188, 84.588, 19.952, -295]
  MoveL 3173 to (46.64, 38.31, -206.02) mm, rotated rx 105.8 ry 33.04 rz -145.95 deg; joints [-8.077, -25.887, 98.043, 143.186, 84.603, 19.942, -295]
  MoveL 3174 to (48.05, 36.82, -206.12) mm, rotated rx 105.8 ry 33.04 rz -145.95 deg; joints [-8.08, -25.75, 97.919, 143.184, 84.614, 19.935, -295]
  MoveL 3175 to (49.52, 35.43, -206.33) mm, rotated rx 105.8 ry 33.04 rz -145.95 deg; joints [-8.086, -25.614, 97.787, 143.177, 84.619, 19.934, -295]
  MoveL 3176 to (51.17, 33.55, -206.47) mm, rotated rx 105.8 ry 33.04 rz -145.95 deg; joints [-8.091, -25.447, 97.642, 143.174, 84.637, 19.923, -295]
  MoveL 3177 to (52.68, 31.63, -206.55) mm, rotated rx 105.8 ry 33.04 rz -145.95 deg; joints [-8.093, -25.286, 97.51, 143.173, 84.661, 19.905, -295]
  MoveL 3178 to (54.14, 29.87, -206.58) mm, rotated rx 105.8 ry 33.04 rz -145.95 deg; joints [-8.094, -25.135, 97.381, 143.174, 84.679, 19.892, -295]
  MoveL 3179 to (55.5, 28.33, -206.63) mm, rotated rx 105.8 ry 33.04 rz -145.95 deg; joints [-8.095, -24.998, 97.261, 143.174, 84.692, 19.882, -295]
  MoveL 3180 to (56.8, 26.86, -206.75) mm, rotated rx 105.8 ry 33.04 rz -145.95 deg; joints [-8.098, -24.867, 97.145, 143.171, 84.705, 19.874, -295]
  MoveL 3181 to (58.15, 25.35, -206.81) mm, rotated rx 105.8 ry 33.04 rz -145.95 deg; joints [-8.1, -24.732, 97.024, 143.171, 84.717, 19.866, -295]
  MoveL 3182 to (59.55, 23.75, -206.88) mm, rotated rx 105.8 ry 33.04 rz -145.95 deg; joints [-8.102, -24.59, 96.898, 143.17, 84.73, 19.857, -295]
  MoveL 3183 to (60.85, 22.25, -207.06) mm, rotated rx 105.8 ry 33.04 rz -145.95 deg; joints [-8.108, -24.458, 96.781, 143.164, 84.743, 19.849, -295]
  MoveL 3184 to (62.08, 20.79, -207.38) mm, rotated rx 105.8 ry 33.04 rz -145.95 deg; joints [-8.12, -24.331, 96.67, 143.154, 84.758, 19.843, -295]
  MoveL 3185 to (62.23, 19.94, -208.42) mm, rotated rx 105.8 ry 33.04 rz -145.95 deg; joints [-8.16, -24.285, 96.656, 143.117, 84.79, 19.833, -295]
  MoveL 3186 to (62.02, 20.09, -208.94) mm, rotated rx 105.8 ry 33.04 rz -145.95 deg; joints [-8.179, -24.302, 96.672, 143.098, 84.794, 19.838, -295]
  MoveL 3187 to (62, 20.08, -209.26) mm, rotated rx 105.8 ry 33.04 rz -145.95 deg; joints [-8.192, -24.302, 96.673, 143.085, 84.796, 19.841, -295]
  MoveL 3188 to (62.15, 19.93, -209.42) mm, rotated rx 105.8 ry 33.04 rz -145.95 deg; joints [-8.198, -24.287, 96.658, 143.08, 84.797, 19.843, -295]
  MoveL 3189 to (62.5, 19.69, -209.46) mm, rotated rx 105.8 ry 33.04 rz -145.95 deg; joints [-8.199, -24.259, 96.625, 143.078, 84.793, 19.846, -295]
  MoveL 3190 to (62.96, 19.45, -209.48) mm, rotated rx 105.8 ry 33.04 rz -145.95 deg; joints [-8.199, -24.225, 96.581, 143.078, 84.786, 19.851, -295]
  MoveL 3191 to (63.52, 19.24, -209.49) mm, rotated rx 105.8 ry 33.04 rz -145.95 deg; joints [-8.198, -24.186, 96.527, 143.078, 84.774, 19.86, -295]
  MoveL 3192 to (64.12, 19.05, -209.5) mm, rotated rx 105.8 ry 33.04 rz -145.95 deg; joints [-8.198, -24.147, 96.47, 143.077, 84.759, 19.871, -295]
  MoveL 3193 to (67.67, 18.14, -209.5) mm, rotated rx 105.8 ry 33.04 rz -145.95 deg; joints [-8.192, -23.922, 96.125, 143.076, 84.661, 19.943, -295]
  MoveL 3194 to (68.09, 18.01, -209.53) mm, rotated rx 105.8 ry 33.04 rz -145.95 deg; joints [-8.192, -23.895, 96.083, 143.075, 84.65, 19.951, -295]
  MoveL 3195 to (68.56, 17.89, -209.54) mm, rotated rx 105.8 ry 33.04 rz -145.95 deg; joints [-8.191, -23.865, 96.037, 143.075, 84.638, 19.96, -295]
  MoveL 3196 to (69.07, 17.75, -209.54) mm, rotated rx 105.8 ry 33.04 rz -145.95 deg; joints [-8.191, -23.833, 95.988, 143.074, 84.624, 19.971, -295]
  MoveL 3197 to (69.54, 17.62, -209.56) mm, rotated rx 105.8 ry 33.04 rz -145.95 deg; joints [-8.191, -23.802, 95.942, 143.074, 84.612, 19.98, -295]
  MoveL 3198 to (69.98, 17.47, -209.6) mm, rotated rx 105.8 ry 33.04 rz -145.95 deg; joints [-8.191, -23.773, 95.899, 143.072, 84.601, 19.988, -295]
  MoveL 3199 to (70.39, 17.33, -209.66) mm, rotated rx 105.8 ry 33.04 rz -145.95 deg; joints [-8.193, -23.745, 95.86, 143.07, 84.591, 19.996, -295]
  MoveL 3200 to (70.84, 17.19, -209.69) mm, rotated rx 105.8 ry 33.04 rz -145.95 deg; joints [-8.194, -23.716, 95.816, 143.069, 84.58, 20.005, -295]
  MoveL 3201 to (71.3, 17.05, -209.71) mm, rotated rx 105.8 ry 33.04 rz -145.95 deg; joints [-8.193, -23.685, 95.77, 143.068, 84.568, 20.014, -295]
  MoveL 3202 to (71.79, 16.92, -209.72) mm, rotated rx 105.8 ry 33.04 rz -145.95 deg; joints [-8.193, -23.654, 95.722, 143.068, 84.554, 20.024, -295]
  MoveL 3203 to (72.3, 16.79, -209.72) mm, rotated rx 105.8 ry 33.04 rz -145.95 deg; joints [-8.192, -23.622, 95.673, 143.067, 84.54, 20.034, -295]
  MoveL 3204 to (75.04, 15.79, -210.06) mm, rotated rx 105.8 ry 33.04 rz -145.95 deg; joints [-8.201, -23.435, 95.404, 143.054, 84.477, 20.085, -295]
  MoveL 3205 to (76.16, 15.13, -210.49) mm, rotated rx 105.8 ry 33.04 rz -145.95 deg; joints [-8.215, -23.347, 95.295, 143.039, 84.462, 20.102, -295]
  MoveL 3206 to (77.11, 14.36, -211.1) mm, rotated rx 105.8 ry 33.04 rz -145.95 deg; joints [-8.237, -23.264, 95.201, 143.017, 84.458, 20.114, -295]
  MoveL 3207 to (78.52, 12.51, -212.83) mm, rotated rx 105.8 ry 33.04 rz -145.95 deg; joints [-8.302, -23.108, 95.064, 142.955, 84.484, 20.119, -295]
  MoveL 3208 to (79.26, 10.22, -215.25) mm, rotated rx 105.8 ry 33.04 rz -145.95 deg; joints [-8.394, -22.969, 94.991, 142.869, 84.555, 20.101, -295]
  MoveL 3209 to (79.24, 8.19, -217.68) mm, rotated rx 105.8 ry 33.04 rz -145.95 deg; joints [-8.488, -22.879, 94.992, 142.783, 84.645, 20.07, -295]
  MoveL 3210 to (78.92, 7.51, -218.63) mm, rotated rx 105.8 ry 33.04 rz -145.95 deg; joints [-8.525, -22.865, 95.023, 142.749, 84.687, 20.052, -295]
  MoveL 3211 to (78.39, 7.07, -219.41) mm, rotated rx 105.8 ry 33.04 rz -145.95 deg; joints [-8.556, -22.873, 95.074, 142.721, 84.728, 20.033, -295]
  MoveL 3212 to (78.04, 6.93, -219.73) mm, rotated rx 105.8 ry 33.04 rz -145.95 deg; joints [-8.569, -22.885, 95.108, 142.709, 84.747, 20.023, -295]
  MoveL 3213 to (77.65, 6.85, -220.01) mm, rotated rx 105.8 ry 33.04 rz -145.95 deg; joints [-8.581, -22.902, 95.146, 142.699, 84.767, 20.012, -295]
  MoveL 3214 to (76.7, 6.86, -220.45) mm, rotated rx 105.8 ry 33.04 rz -145.95 deg; joints [-8.599, -22.951, 95.239, 142.684, 84.804, 19.991, -295]
  MoveL 3215 to (75.54, 7.1, -220.71) mm, rotated rx 105.8 ry 33.04 rz -145.95 deg; joints [-8.611, -23.022, 95.352, 142.674, 84.84, 19.968, -295]
  MoveL 3216 to (74.16, 7.57, -220.79) mm, rotated rx 105.8 ry 33.04 rz -145.95 deg; joints [-8.617, -23.114, 95.485, 142.671, 84.874, 19.944, -295]
  MoveL 3217 to (73.68, 7.77, -220.79) mm, rotated rx 105.8 ry 33.04 rz -145.95 deg; joints [-8.618, -23.147, 95.532, 142.671, 84.885, 19.936, -295]
  MoveL 3218 to (73.26, 7.95, -220.76) mm, rotated rx 105.8 ry 33.04 rz -145.95 deg; joints [-8.618, -23.177, 95.573, 142.672, 84.894, 19.929, -295]
  MoveL 3219 to (72.88, 8.14, -220.72) mm, rotated rx 105.8 ry 33.04 rz -145.95 deg; joints [-8.617, -23.205, 95.61, 142.673, 84.901, 19.923, -295]
  MoveL 3220 to (72.5, 8.34, -220.66) mm, rotated rx 105.8 ry 33.04 rz -145.95 deg; joints [-8.615, -23.234, 95.647, 142.675, 84.907, 19.918, -295]
  MoveL 3221 to (72.09, 8.53, -220.62) mm, rotated rx 105.8 ry 33.04 rz -145.95 deg; joints [-8.614, -23.263, 95.686, 142.677, 84.915, 19.912, -295]
  MoveL 3222 to (71.62, 8.73, -220.6) mm, rotated rx 105.8 ry 33.04 rz -145.95 deg; joints [-8.614, -23.296, 95.732, 142.677, 84.925, 19.904, -295]
  MoveL 3223 to (71.14, 8.92, -220.6) mm, rotated rx 105.8 ry 33.04 rz -145.95 deg; joints [-8.615, -23.33, 95.779, 142.677, 84.936, 19.896, -295]
  MoveL 3224 to (70.67, 9.11, -220.6) mm, rotated rx 105.8 ry 33.04 rz -145.95 deg; joints [-8.616, -23.362, 95.824, 142.677, 84.946, 19.888, -295]
  MoveL 3225 to (70.24, 9.3, -220.57) mm, rotated rx 105.8 ry 33.04 rz -145.95 deg; joints [-8.616, -23.393, 95.866, 142.678, 84.955, 19.881, -295]
  MoveL 3226 to (69.86, 9.48, -220.52) mm, rotated rx 105.8 ry 33.04 rz -145.95 deg; joints [-8.614, -23.421, 95.904, 142.68, 84.962, 19.875, -295]
  MoveL 3227 to (69.48, 9.66, -220.46) mm, rotated rx 105.8 ry 33.04 rz -145.95 deg; joints [-8.613, -23.449, 95.94, 142.682, 84.969, 19.869, -295]
  MoveL 3228 to (69.06, 9.87, -220.4) mm, rotated rx 105.8 ry 33.04 rz -145.95 deg; joints [-8.611, -23.479, 95.981, 142.684, 84.977, 19.863, -295]
  MoveL 3229 to (68.49, 10.12, -220.37) mm, rotated rx 105.8 ry 33.04 rz -145.95 deg; joints [-8.611, -23.52, 96.035, 142.685, 84.988, 19.854, -295]
  MoveL 3230 to (67.77, 10.44, -220.35) mm, rotated rx 105.8 ry 33.04 rz -145.95 deg; joints [-8.611, -23.571, 96.105, 142.685, 85.003, 19.843, -295]
  MoveL 3231 to (66.31, 11.02, -220.35) mm, rotated rx 105.8 ry 33.04 rz -145.95 deg; joints [-8.614, -23.672, 96.246, 142.685, 85.035, 19.819, -295]
  MoveL 3232 to (65.54, 11.33, -220.32) mm, rotated rx 105.8 ry 33.04 rz -145.95 deg; joints [-8.614, -23.726, 96.32, 142.686, 85.051, 19.807, -295]
  MoveL 3233 to (64.96, 11.58, -220.3) mm, rotated rx 105.8 ry 33.04 rz -145.95 deg; joints [-8.615, -23.766, 96.376, 142.686, 85.063, 19.798, -295]
  MoveL 3234 to (64.53, 11.8, -220.3) mm, rotated rx 105.8 ry 33.04 rz -145.95 deg; joints [-8.615, -23.798, 96.417, 142.686, 85.071, 19.793, -295]
  MoveL 3235 to (64.18, 12.03, -220.28) mm, rotated rx 105.8 ry 33.04 rz -145.95 deg; joints [-8.615, -23.826, 96.451, 142.687, 85.075, 19.789, -295]
  MoveL 3236 to (64.03, 12.18, -220.17) mm, rotated rx 105.8 ry 33.04 rz -145.95 deg; joints [-8.611, -23.841, 96.465, 142.691, 85.074, 19.788, -295]
  MoveL 3237 to (64.1, 12.18, -219.95) mm, rotated rx 105.8 ry 33.04 rz -145.95 deg; joints [-8.602, -23.837, 96.459, 142.699, 85.071, 19.788, -295]
  MoveL 3238 to (64.4, 12.02, -219.6) mm, rotated rx 105.8 ry 33.04 rz -145.95 deg; joints [-8.589, -23.816, 96.433, 142.712, 85.065, 19.787, -295]
  MoveL 3239 to (64.46, 12.8, -218.9) mm, rotated rx 105.8 ry 33.04 rz -145.95 deg; joints [-8.561, -23.847, 96.426, 142.737, 85.029, 19.804, -295]
  MoveL 3240 to (63.35, 14.48, -218.75) mm, rotated rx 105.8 ry 33.04 rz -145.95 deg; joints [-8.555, -23.977, 96.525, 142.741, 85.003, 19.822, -295]
  MoveL 3241 to (62.32, 16.11, -218.46) mm, rotated rx 105.8 ry 33.04 rz -145.95 deg; joints [-8.545, -24.101, 96.616, 142.749, 84.975, 19.839, -295]
  MoveL 3242 to (61.27, 17.72, -218.19) mm, rotated rx 105.8 ry 33.04 rz -145.95 deg; joints [-8.534, -24.226, 96.71, 142.758, 84.949, 19.855, -295]
  MoveL 3243 to (60.21, 19.34, -217.92) mm, rotated rx 105.8 ry 33.04 rz -145.95 deg; joints [-8.524, -24.351, 96.804, 142.766, 84.922, 19.872, -295]
  MoveL 3244 to (59.09, 21.03, -217.7) mm, rotated rx 105.8 ry 33.04 rz -145.95 deg; joints [-8.516, -24.482, 96.902, 142.772, 84.894, 19.89, -295]
  MoveL 3245 to (57.98, 22.84, -217.56) mm, rotated rx 105.8 ry 33.04 rz -145.95 deg; joints [-8.511, -24.618, 96.998, 142.775, 84.862, 19.912, -295]
  MoveL 3246 to (56.74, 25.05, -217.45) mm, rotated rx 105.8 ry 33.04 rz -145.95 deg; joints [-8.507, -24.777, 97.103, 142.776, 84.818, 19.945, -295]
  MoveL 3247 to (55.22, 27.02, -217.38) mm, rotated rx 105.8 ry 33.04 rz -145.95 deg; joints [-8.504, -24.941, 97.236, 142.777, 84.793, 19.963, -295]
  MoveL 3248 to (53.94, 28.7, -217.26) mm, rotated rx 105.8 ry 33.04 rz -145.95 deg; joints [-8.501, -25.08, 97.349, 142.779, 84.772, 19.978, -295]
  MoveL 3249 to (52.83, 30.23, -217.09) mm, rotated rx 105.8 ry 33.04 rz -145.95 deg; joints [-8.494, -25.204, 97.446, 142.783, 84.749, 19.992, -295]
  MoveL 3250 to (51.66, 31.91, -216.96) mm, rotated rx 105.8 ry 33.04 rz -145.95 deg; joints [-8.49, -25.336, 97.547, 142.786, 84.723, 20.011, -295]
  MoveL 3251 to (50.48, 33.62, -216.83) mm, rotated rx 105.8 ry 33.04 rz -145.95 deg; joints [-8.485, -25.472, 97.648, 142.789, 84.695, 20.03, -295]
  MoveL 3252 to (49.24, 35.41, -216.76) mm, rotated rx 105.8 ry 33.04 rz -145.95 deg; joints [-8.483, -25.612, 97.753, 142.789, 84.666, 20.051, -295]
  MoveL 3253 to (48.02, 37.16, -216.53) mm, rotated rx 105.8 ry 33.04 rz -145.95 deg; joints [-8.475, -25.751, 97.858, 142.795, 84.638, 20.07, -295]
  MoveL 3254 to (46.8, 38.92, -216.42) mm, rotated rx 105.8 ry 33.04 rz -145.95 deg; joints [-8.471, -25.89, 97.961, 142.797, 84.609, 20.09, -295]
  MoveL 3255 to (45.57, 40.66, -216.2) mm, rotated rx 105.8 ry 33.04 rz -145.95 deg; joints [-8.463, -26.028, 98.066, 142.803, 84.58, 20.109, -295]
  MoveL 3256 to (44.35, 42.41, -216.09) mm, rotated rx 105.8 ry 33.04 rz -145.95 deg; joints [-8.459, -26.167, 98.169, 142.805, 84.551, 20.129, -295]
  MoveL 3257 to (43.11, 44.15, -215.87) mm, rotated rx 105.8 ry 33.04 rz -145.95 deg; joints [-8.451, -26.306, 98.275, 142.81, 84.523, 20.148, -295]
  MoveL 3258 to (41.88, 45.89, -215.76) mm, rotated rx 105.8 ry 33.04 rz -145.95 deg; joints [-8.447, -26.445, 98.377, 142.812, 84.494, 20.169, -295]
  MoveL 3259 to (40.65, 47.64, -215.65) mm, rotated rx 105.8 ry 33.04 rz -145.95 deg; joints [-8.443, -26.583, 98.48, 142.813, 84.464, 20.19, -295]
  MoveL 3260 to (39.5, 49.17, -215.42) mm, rotated rx 105.8 ry 33.04 rz -145.95 deg; joints [-8.435, -26.709, 98.578, 142.82, 84.44, 20.205, -295]
  MoveL 3261 to (38.37, 50.61, -215.12) mm, rotated rx 105.8 ry 33.04 rz -145.95 deg; joints [-8.424, -26.829, 98.674, 142.829, 84.419, 20.216, -295]
  MoveL 3262 to (37.22, 51.99, -214.73) mm, rotated rx 105.8 ry 33.04 rz -145.95 deg; joints [-8.41, -26.949, 98.774, 142.842, 84.401, 20.225, -295]
  MoveL 3263 to (37.78, 50.69, -213.81) mm, rotated rx 105.8 ry 33.04 rz -145.95 deg; joints [-8.375, -26.866, 98.738, 142.878, 84.432, 20.187, -295]
  MoveL 3264 to (37.58, 51, -213.75) mm, rotated rx 105.8 ry 33.04 rz -145.95 deg; joints [-8.373, -26.889, 98.755, 142.88, 84.426, 20.191, -295]
  MoveL 3265 to (37.41, 51.32, -213.69) mm, rotated rx 105.8 ry 33.04 rz -145.95 deg; joints [-8.371, -26.912, 98.769, 142.882, 84.419, 20.196, -295]
  MoveL 3266 to (37.28, 51.72, -213.66) mm, rotated rx 105.8 ry 33.04 rz -145.95 deg; joints [-8.369, -26.936, 98.777, 142.882, 84.406, 20.205, -295]
  MoveL 3267 to (37.2, 52.16, -213.63) mm, rotated rx 105.8 ry 33.04 rz -145.95 deg; joints [-8.368, -26.959, 98.781, 142.883, 84.391, 20.216, -295]
  MoveL 3268 to (37.16, 52.66, -213.63) mm, rotated rx 105.8 ry 33.04 rz -145.95 deg; joints [-8.367, -26.982, 98.779, 142.882, 84.371, 20.231, -295]
  MoveL 3269 to (37.14, 53.18, -213.62) mm, rotated rx 105.8 ry 33.04 rz -145.95 deg; joints [-8.366, -27.005, 98.776, 142.881, 84.349, 20.247, -295]
  MoveL 3270 to (37.13, 54.23, -213.62) mm, rotated rx 105.8 ry 33.04 rz -145.95 deg; joints [-8.365, -27.05, 98.766, 142.879, 84.305, 20.28, -295]
  MoveL 3271 to (37.11, 54.72, -213.6) mm, rotated rx 105.8 ry 33.04 rz -145.95 deg; joints [-8.364, -27.072, 98.763, 142.879, 84.285, 20.294, -295]
  MoveL 3272 to (37.07, 55.18, -213.56) mm, rotated rx 105.8 ry 33.04 rz -145.95 deg; joints [-8.361, -27.093, 98.762, 142.88, 84.267, 20.308, -295]
  MoveL 3273 to (37.01, 55.7, -213.48) mm, rotated rx 105.8 ry 33.04 rz -145.95 deg; joints [-8.358, -27.119, 98.763, 142.882, 84.247, 20.322, -295]
  MoveL 3274 to (36.96, 56.28, -213.41) mm, rotated rx 105.8 ry 33.04 rz -145.95 deg; joints [-8.354, -27.146, 98.762, 142.883, 84.224, 20.338, -295]
  MoveL 3275 to (36.93, 56.86, -213.38) mm, rotated rx 105.8 ry 33.04 rz -145.95 deg; joints [-8.352, -27.171, 98.758, 142.883, 84.2, 20.355, -295]
  MoveL 3276 to (36.92, 57.4, -213.37) mm, rotated rx 105.8 ry 33.04 rz -145.95 deg; joints [-8.351, -27.195, 98.754, 142.883, 84.178, 20.371, -295]
  MoveL 3277 to (36.91, 57.93, -213.36) mm, rotated rx 105.8 ry 33.04 rz -145.95 deg; joints [-8.351, -27.218, 98.749, 142.882, 84.155, 20.388, -295]
  MoveL 3278 to (36.9, 58.98, -213.36) mm, rotated rx 105.8 ry 33.04 rz -145.95 deg; joints [-8.349, -27.262, 98.739, 142.88, 84.111, 20.421, -295]
  MoveL 3279 to (36.85, 60.01, -213.34) mm, rotated rx 105.8 ry 33.04 rz -145.95 deg; joints [-8.347, -27.308, 98.732, 142.879, 84.07, 20.452, -295]
  MoveL 3280 to (36.82, 62.63, -213.34) mm, rotated rx 105.8 ry 33.04 rz -145.95 deg; joints [-8.343, -27.419, 98.706, 142.874, 83.96, 20.534, -295]
  MoveL 3281 to (36.87, 64.07, -213.43) mm, rotated rx 105.8 ry 33.04 rz -145.95 deg; joints [-8.345, -27.477, 98.685, 142.867, 83.897, 20.583, -295]
  MoveL 3282 to (37.05, 65.24, -213.69) mm, rotated rx 105.8 ry 33.04 rz -145.95 deg; joints [-8.353, -27.515, 98.652, 142.855, 83.842, 20.628, -295]
  MoveL 3283 to (37.38, 66.12, -214.13) mm, rotated rx 105.8 ry 33.04 rz -145.95 deg; joints [-8.367, -27.534, 98.608, 142.836, 83.794, 20.67, -295]
  MoveL 3284 to (37.6, 66.46, -214.41) mm, rotated rx 105.8 ry 33.04 rz -145.95 deg; joints [-8.377, -27.536, 98.581, 142.825, 83.773, 20.69, -295]
  MoveL 3285 to (37.84, 66.72, -214.74) mm, rotated rx 105.8 ry 33.04 rz -145.95 deg; joints [-8.389, -27.533, 98.552, 142.812, 83.755, 20.709, -295]
  MoveL 3286 to (38.45, 67.04, -215.53) mm, rotated rx 105.8 ry 33.04 rz -145.95 deg; joints [-8.417, -27.513, 98.486, 142.781, 83.723, 20.745, -295]
  MoveL 3287 to (39.19, 67.08, -216.5) mm, rotated rx 105.8 ry 33.04 rz -145.95 deg; joints [-8.452, -27.474, 98.408, 142.745, 83.699, 20.777, -295]
  MoveL 3288 to (41.08, 66.3, -218.95) mm, rotated rx 105.8 ry 33.04 rz -145.95 deg; joints [-8.542, -27.337, 98.218, 142.654, 83.675, 20.833, -295]
